LIN {X 0,Y 450.546,Z 601.299,A -85,B 0,C 180,E1 -16151.951,E2 -16151.951} C_VEL
LIN {X 0,Y 450.573,Z 601.291,A -85,B 0,C 180,E1 -16154.391,E2 -16154.391} C_VEL
LIN {X 0,Y 450.568,Z 601.288,A -85,B 0,C 180,E1 -16156.941,E2 -16156.941} C_VEL
LIN {X 0,Y 450.573,Z 601.291,A -85,B 0,C 180,E1 -16160.405,E2 -16160.405} C_VEL
LIN {X 0,Y 450.592,Z 601.291,A -85,B 0,C 180,E1 -16163.793,E2 -16163.793} C_VEL
LIN {X 0,Y 450.566,Z 601.289,A -85,B 0,C 180,E1 -16167.085,E2 -16167.085} C_VEL
LIN {X 0,Y 450.558,Z 601.295,A -85,B 0,C 180,E1 -16170.167,E2 -16170.167} C_VEL
LIN {X 0,Y 450.589,Z 601.286,A -85,B 0,C 180,E1 -16173.205,E2 -16173.205} C_VEL
LIN {X 0,Y 450.58,Z 601.289,A -85,B 0,C 180,E1 -16176.517,E2 -16176.517} C_VEL
LIN {X 0,Y 450.593,Z 601.293,A -85,B 0,C 180,E1 -16180.002,E2 -16180.002} C_VEL
LIN {X 0,Y 450.589,Z 601.286,A -85,B 0,C 180,E1 -16182.821,E2 -16182.821} C_VEL
LIN {X 0,Y 450.626,Z 601.284,A -85,B 0,C 180,E1 -16185.6,E2 -16185.6} C_VEL
LIN {X 0,Y 450.749,Z 601.269,A -85,B 0,C 180,E1 -16188.346,E2 -16188.346} C_VEL
LIN {X 0,Y 450.78,Z 601.27,A -85,B 0,C 180,E1 -16191.961,E2 -16191.961} C_VEL
LIN {X 0,Y 450.913,Z 601.251,A -85,B 0,C 180,E1 -16193.81,E2 -16193.81} C_VEL
LIN {X 0,Y 450.837,Z 601.258,A -85,B 0,C 180,E1 -16196.437,E2 -16196.437} C_VEL
LIN {X 0,Y 450.905,Z 601.254,A -85,B 0,C 180,E1 -16200,E2 -16200} C_VEL
LIN {X 0,Y 450.866,Z 601.254,A -85,B 0,C 180,E1 -16204.455,E2 -16204.455} C_VEL
LIN {X 0,Y 450.774,Z 601.263,A -85,B 0,C 180,E1 -16207.141,E2 -16207.141} C_VEL
LIN {X 0,Y 450.679,Z 601.281,A -85,B 0,C 180,E1 -16209.844,E2 -16209.844} C_VEL
LIN {X 0,Y 450.674,Z 601.277,A -85,B 0,C 180,E1 -16212.568,E2 -16212.568} C_VEL
LIN {X 0,Y 450.622,Z 601.284,A -85,B 0,C 180,E1 -16215.48,E2 -16215.48} C_VEL
LIN {X 0,Y 450.567,Z 601.289,A -85,B 0,C 180,E1 -16219.054,E2 -16219.054} C_VEL
LIN {X 0,Y 450.548,Z 601.298,A -85,B 0,C 180,E1 -16221.908,E2 -16221.908} C_VEL
LIN {X 0,Y 450.531,Z 601.293,A -85,B 0,C 180,E1 -16224.82,E2 -16224.82} C_VEL
LIN {X 0,Y 450.577,Z 601.293,A -85,B 0,C 180,E1 -16227.799,E2 -16227.799} C_VEL
LIN {X 0,Y 450.517,Z 601.295,A -85,B 0,C 180,E1 -16230.869,E2 -16230.869} C_VEL
LIN {X 0,Y 450.532,Z 601.3,A -85,B 0,C 180,E1 -16234.035,E2 -16234.035} C_VEL
LIN {X 0,Y 450.534,Z 601.298,A -85,B 0,C 180,E1 -16236.213,E2 -16236.213} C_VEL
LIN {X 0,Y 450.5,Z 601.3,A -85,B 0,C 180,E1 -16239.604,E2 -16239.604} C_VEL
LIN {X 0,Y 450.53,Z 601.301,A -85,B 0,C 180,E1 -16241.953,E2 -16241.953} C_VEL
LIN {X 0,Y 450.556,Z 601.293,A -85,B 0,C 180,E1 -16244.393,E2 -16244.393} C_VEL
LIN {X 0,Y 450.538,Z 601.292,A -85,B 0,C 180,E1 -16246.945,E2 -16246.945} C_VEL
LIN {X 0,Y 450.509,Z 601.299,A -85,B 0,C 180,E1 -16249.627,E2 -16249.627} C_VEL
LIN {X 0,Y 450.48,Z 601.3,A -85,B 0,C 180,E1 -16252.67,E2 -16252.67} C_VEL
LIN {X 0,Y 450.521,Z 601.302,A -85,B 0,C 180,E1 -16255.965,E2 -16255.965} C_VEL
LIN {X 0,Y 450.517,Z 601.295,A -85,B 0,C 180,E1 -16259.132,E2 -16259.132} C_VEL
LIN {X 0,Y 450.547,Z 601.291,A -85,B 0,C 180,E1 -16261.188,E2 -16261.188} C_VEL
LIN {X 0,Y 450.616,Z 601.459,A -85,B 0,C 180,E1 -16264.463,E2 -16264.463} C_VEL
LIN {X 0,Y 453.094,Z 615.734,A -85,B 0,C 180,E1 -16267.528,E2 -16267.528} C_VEL
LIN {X 0,Y 452.123,Z 628.307,A -85,B 0,C 180,E1 -16270.073,E2 -16270.073} C_VEL
LIN {X 0,Y 450.856,Z 645.268,A -85,B 0,C 180,E1 -16273.471,E2 -16273.471} C_VEL
LIN {X 0,Y 453.98,Z 674.168,A -85,B 0,C 180,E1 -16274.153,E2 -16274.153} C_VEL
LIN {X 0,Y 454.049,Z 687.401,A -85,B 0,C 180,E1 -16274.424,E2 -16274.424} C_VEL
LIN {X 0,Y 452.771,Z 752.366,A -85,B 0,C 180,E1 -16275.726,E2 -16275.726} C_VEL
LIN {X 0,Y 452.55,Z 762.586,A -85,B 0,C 180,E1 -16276.034,E2 -16276.034} C_VEL
LIN {X 0,Y 452.15,Z 772.789,A -85,B 0,C 180,E1 -16276.449,E2 -16276.449} C_VEL
LIN {X 0,Y 451.855,Z 781.497,A -85,B 0,C 180,E1 -16276.897,E2 -16276.897} C_VEL
LIN {X 0,Y 451.313,Z 791.921,A -85,B 0,C 180,E1 -16277.565,E2 -16277.565} C_VEL
LIN {X 0,Y 450.749,Z 801.808,A -85,B 0,C 180,E1 -16278.345,E2 -16278.345} C_VEL
LIN {X 0,Y 450.383,Z 810.122,A -85,B 0,C 180,E1 -16279.131,E2 -16279.131} C_VEL
LIN {X 0,Y 449.846,Z 819.008,A -85,B 0,C 180,E1 -16280.138,E2 -16280.138} C_VEL
LIN {X 0,Y 449.477,Z 825.737,A -85,B 0,C 180,E1 -16281.035,E2 -16281.035} C_VEL
LIN {X 0,Y 449.096,Z 832.781,A -85,B 0,C 180,E1 -16282.156,E2 -16282.156} C_VEL
LIN {X 0,Y 448.876,Z 838.658,A -85,B 0,C 180,E1 -16283.279,E2 -16283.279} C_VEL
LIN {X 0,Y 448.702,Z 844.329,A -85,B 0,C 180,E1 -16284.626,E2 -16284.626} C_VEL
LIN {X 0,Y 448.577,Z 848.751,A -85,B 0,C 180,E1 -16285.971,E2 -16285.971} C_VEL
LIN {X 0,Y 448.542,Z 852.046,A -85,B 0,C 180,E1 -16287.315,E2 -16287.315} C_VEL
LIN {X 0,Y 448.542,Z 853.712,A -85,B 0,C 180,E1 -16288.21,E2 -16288.21} C_VEL
LIN {X 0,Y 448.535,Z 855.564,A -85,B 0,C 180,E1 -16290,E2 -16290} C_VEL
LIN {X 0,Y 448.515,Z 855.863,A -85,B 0,C 180,E1 -16290.895,E2 -16290.895} C_VEL
LIN {X 0,Y 448.491,Z 855.194,A -85,B 0,C 180,E1 -16292.686,E2 -16292.686} C_VEL
LIN {X 0,Y 448.542,Z 854.146,A -85,B 0,C 180,E1 -16293.581,E2 -16293.581} C_VEL
LIN {X 0,Y 448.749,Z 850.921,A -85,B 0,C 180,E1 -16295.374,E2 -16295.374} C_VEL
LIN {X 0,Y 449.026,Z 847.231,A -85,B 0,C 180,E1 -16296.719,E2 -16296.719} C_VEL
LIN {X 0,Y 449.487,Z 842.395,A -85,B 0,C 180,E1 -16298.062,E2 -16298.062} C_VEL
LIN {X 0,Y 450.082,Z 836.291,A -85,B 0,C 180,E1 -16299.405,E2 -16299.405} C_VEL
LIN {X 0,Y 450.945,Z 828.69,A -85,B 0,C 180,E1 -16300.743,E2 -16300.743} C_VEL
LIN {X 0,Y 451.886,Z 821.013,A -85,B 0,C 180,E1 -16301.852,E2 -16301.852} C_VEL
LIN {X 0,Y 452.624,Z 813.883,A -85,B 0,C 180,E1 -16302.731,E2 -16302.731} C_VEL
LIN {X 0,Y 453.681,Z 804.065,A -85,B 0,C 180,E1 -16303.732,E2 -16303.732} C_VEL
LIN {X 0,Y 454.54,Z 795.005,A -85,B 0,C 180,E1 -16304.502,E2 -16304.502} C_VEL
LIN {X 0,Y 455.414,Z 785.704,A -85,B 0,C 180,E1 -16305.157,E2 -16305.157} C_VEL
LIN {X 0,Y 456.23,Z 775.218,A -85,B 0,C 180,E1 -16305.757,E2 -16305.757} C_VEL
LIN {X 0,Y 457.128,Z 763.471,A -85,B 0,C 180,E1 -16306.267,E2 -16306.267} C_VEL
LIN {X 0,Y 457.765,Z 752.645,A -85,B 0,C 180,E1 -16306.616,E2 -16306.616} C_VEL
LIN {X 0,Y 458.823,Z 722.033,A -85,B 0,C 180,E1 -16307.29,E2 -16307.29} C_VEL
LIN {X 0,Y 460.202,Z 677.981,A -85,B 0,C 180,E1 -16308.254,E2 -16308.254} C_VEL
LIN {X 0,Y 457.656,Z 661.739,A -85,B 0,C 180,E1 -16308.813,E2 -16308.813} C_VEL
LIN {X 0,Y 454.289,Z 646.219,A -85,B 0,C 180,E1 -16309.435,E2 -16309.435} C_VEL
LIN {X 0,Y 453.659,Z 643.473,A -85,B 0,C 180,E1 -16309.562,E2 -16309.562} C_VEL
LIN {X 0,Y 455.818,Z 627.583,A -85,B 0,C 180,E1 -16313.07,E2 -16313.07} C_VEL
LIN {X 0,Y 454.965,Z 621.055,A -85,B 0,C 180,E1 -16314.723,E2 -16314.723} C_VEL
LIN {X 0,Y 453.262,Z 612.283,A -85,B 0,C 180,E1 -16317.122,E2 -16317.122} C_VEL
LIN {X 0,Y 451.108,Z 603.423,A -85,B 0,C 180,E1 -16319.793,E2 -16319.793} C_VEL
LIN {X 0,Y 450.552,Z 601.297,A -85,B 0,C 180,E1 -16320.478,E2 -16320.478} C_VEL
LIN {X 0,Y 450.545,Z 601.297,A -85,B 0,C 180,E1 -16324.034,E2 -16324.034} C_VEL
LIN {X 0,Y 450.52,Z 601.296,A -85,B 0,C 180,E1 -16327.326,E2 -16327.326} C_VEL
LIN {X 0,Y 450.53,Z 601.291,A -85,B 0,C 180,E1 -16330.376,E2 -16330.376} C_VEL
LIN {X 0,Y 450.55,Z 601.291,A -85,B 0,C 180,E1 -16333.161,E2 -16333.161} C_VEL
LIN {X 0,Y 450.576,Z 601.291,A -85,B 0,C 180,E1 -16335.651,E2 -16335.651} C_VEL
LIN {X 0,Y 450.551,Z 601.296,A -85,B 0,C 180,E1 -16338.265,E2 -16338.265} C_VEL
LIN {X 0,Y 450.564,Z 601.292,A -85,B 0,C 180,E1 -16341.014,E2 -16341.014} C_VEL
LIN {X 0,Y 450.555,Z 601.294,A -85,B 0,C 180,E1 -16343.941,E2 -16343.941} C_VEL
LIN {X 0,Y 450.579,Z 601.295,A -85,B 0,C 180,E1 -16347.083,E2 -16347.083} C_VEL
LIN {X 0,Y 450.562,Z 601.292,A -85,B 0,C 180,E1 -16350.167,E2 -16350.167} C_VEL
LIN {X 0,Y 450.602,Z 601.289,A -85,B 0,C 180,E1 -16353.205,E2 -16353.205} C_VEL
LIN {X 0,Y 450.584,Z 601.295,A -85,B 0,C 180,E1 -16356.517,E2 -16356.517} C_VEL
LIN {X 0,Y 450.597,Z 601.297,A -85,B 0,C 180,E1 -16360.002,E2 -16360.002} C_VEL
LIN {X 0,Y 450.61,Z 601.344,A -85,B 0,C 180,E1 -16362.589,E2 -16362.589} C_VEL
LIN {X 0,Y 452.468,Z 609.128,A -85,B 0,C 180,E1 -16365.201,E2 -16365.201} C_VEL
LIN {X 0,Y 454.016,Z 616.689,A -85,B 0,C 180,E1 -16367.526,E2 -16367.526} C_VEL
LIN {X 0,Y 454.947,Z 623.05,A -85,B 0,C 180,E1 -16369.353,E2 -16369.353} C_VEL
LIN {X 0,Y 454.575,Z 627.715,A -85,B 0,C 180,E1 -16370.56,E2 -16370.56} C_VEL
LIN {X 0,Y 459.098,Z 645.694,A -85,B 0,C 180,E1 -16371.343,E2 -16371.343} C_VEL
LIN {X 0,Y 460.909,Z 655.517,A -85,B 0,C 180,E1 -16371.699,E2 -16371.699} C_VEL
LIN {X 0,Y 458.567,Z 715.512,A -85,B 0,C 180,E1 -16372.981,E2 -16372.981} C_VEL
LIN {X 0,Y 457.808,Z 737.352,A -85,B 0,C 180,E1 -16373.493,E2 -16373.493} C_VEL
LIN {X 0,Y 457.027,Z 751.138,A -85,B 0,C 180,E1 -16374.007,E2 -16374.007} C_VEL
LIN {X 0,Y 456.261,Z 762.657,A -85,B 0,C 180,E1 -16374.604,E2 -16374.604} C_VEL
LIN {X 0,Y 455.54,Z 772.672,A -85,B 0,C 180,E1 -16375.259,E2 -16375.259} C_VEL
LIN {X 0,Y 454.727,Z 782.259,A -85,B 0,C 180,E1 -16376.025,E2 -16376.025} C_VEL
LIN {X 0,Y 453.809,Z 791.383,A -85,B 0,C 180,E1 -16376.903,E2 -16376.903} C_VEL
LIN {X 0,Y 452.94,Z 799.112,A -85,B 0,C 180,E1 -16377.784,E2 -16377.784} C_VEL
LIN {X 0,Y 451.916,Z 807.198,A -85,B 0,C 180,E1 -16378.89,E2 -16378.89} C_VEL
LIN {X 0,Y 451.029,Z 813.945,A -85,B 0,C 180,E1 -16380,E2 -16380} C_VEL
LIN {X 0,Y 450.508,Z 818.593,A -85,B 0,C 180,E1 -16380.891,E2 -16380.891} C_VEL
LIN {X 0,Y 449.775,Z 824.257,A -85,B 0,C 180,E1 -16382.231,E2 -16382.231} C_VEL
LIN {X 0,Y 449.416,Z 828.692,A -85,B 0,C 180,E1 -16383.574,E2 -16383.574} C_VEL
LIN {X 0,Y 449.156,Z 831.048,A -85,B 0,C 180,E1 -16384.472,E2 -16384.472} C_VEL
LIN {X 0,Y 448.716,Z 834.413,A -85,B 0,C 180,E1 -16386.273,E2 -16386.273} C_VEL
LIN {X 0,Y 448.549,Z 835.387,A -85,B 0,C 180,E1 -16387.176,E2 -16387.176} C_VEL
LIN {X 0,Y 448.418,Z 836.149,A -85,B 0,C 180,E1 -16388.986,E2 -16388.986} C_VEL
LIN {X 0,Y 448.466,Z 835.598,A -85,B 0,C 180,E1 -16390.269,E2 -16390.269} C_VEL
LIN {X 0,Y 448.381,Z 833.919,A -85,B 0,C 180,E1 -16391.717,E2 -16391.717} C_VEL
LIN {X 0,Y 448.492,Z 831.264,A -85,B 0,C 180,E1 -16393.088,E2 -16393.088} C_VEL
LIN {X 0,Y 448.702,Z 827.132,A -85,B 0,C 180,E1 -16394.567,E2 -16394.567} C_VEL
LIN {X 0,Y 448.922,Z 821.42,A -85,B 0,C 180,E1 -16396.078,E2 -16396.078} C_VEL
LIN {X 0,Y 449.14,Z 815.962,A -85,B 0,C 180,E1 -16397.236,E2 -16397.236} C_VEL
LIN {X 0,Y 449.473,Z 809.329,A -85,B 0,C 180,E1 -16398.395,E2 -16398.395} C_VEL
LIN {X 0,Y 449.829,Z 803.085,A -85,B 0,C 180,E1 -16399.322,E2 -16399.322} C_VEL
LIN {X 0,Y 450.304,Z 793.566,A -85,B 0,C 180,E1 -16400.486,E2 -16400.486} C_VEL
LIN {X 0,Y 450.736,Z 784.964,A -85,B 0,C 180,E1 -16401.362,E2 -16401.362} C_VEL
LIN {X 0,Y 451.211,Z 776.182,A -85,B 0,C 180,E1 -16402.113,E2 -16402.113} C_VEL
LIN {X 0,Y 451.7,Z 766.35,A -85,B 0,C 180,E1 -16402.809,E2 -16402.809} C_VEL
LIN {X 0,Y 452.132,Z 756.214,A -85,B 0,C 180,E1 -16403.389,E2 -16403.389} C_VEL
LIN {X 0,Y 452.394,Z 745.054,A -85,B 0,C 180,E1 -16403.886,E2 -16403.886} C_VEL
LIN {X 0,Y 452.747,Z 734.354,A -85,B 0,C 180,E1 -16404.235,E2 -16404.235} C_VEL
LIN {X 0,Y 453.276,Z 712.839,A -85,B 0,C 180,E1 -16404.69,E2 -16404.69} C_VEL
LIN {X 0,Y 454.432,Z 650.819,A -85,B 0,C 180,E1 -16405.918,E2 -16405.918} C_VEL
LIN {X 0,Y 451.139,Z 625.367,A -85,B 0,C 180,E1 -16406.542,E2 -16406.542} C_VEL
LIN {X 0,Y 452.027,Z 612.321,A -85,B 0,C 180,E1 -16409.471,E2 -16409.471} C_VEL
LIN {X 0,Y 451.77,Z 607.809,A -85,B 0,C 180,E1 -16410.515,E2 -16410.515} C_VEL
LIN {X 0,Y 450.631,Z 601.287,A -85,B 0,C 180,E1 -16412.099,E2 -16412.099} C_VEL
LIN {X 0,Y 450.56,Z 601.289,A -85,B 0,C 180,E1 -16415.113,E2 -16415.113} C_VEL
LIN {X 0,Y 450.547,Z 601.293,A -85,B 0,C 180,E1 -16418.451,E2 -16418.451} C_VEL
LIN {X 0,Y 450.55,Z 601.291,A -85,B 0,C 180,E1 -16420.764,E2 -16420.764} C_VEL
LIN {X 0,Y 450.57,Z 601.288,A -85,B 0,C 180,E1 -16423.157,E2 -16423.157} C_VEL
LIN {X 0,Y 450.574,Z 601.291,A -85,B 0,C 180,E1 -16425.65,E2 -16425.65} C_VEL
LIN {X 0,Y 450.548,Z 601.295,A -85,B 0,C 180,E1 -16428.264,E2 -16428.264} C_VEL
LIN {X 0,Y 450.561,Z 601.289,A -85,B 0,C 180,E1 -16431.013,E2 -16431.013} C_VEL
LIN {X 0,Y 450.578,Z 601.295,A -85,B 0,C 180,E1 -16433.935,E2 -16433.935} C_VEL
LIN {X 0,Y 450.566,Z 601.289,A -85,B 0,C 180,E1 -16437.084,E2 -16437.084} C_VEL
LIN {X 0,Y 450.577,Z 601.289,A -85,B 0,C 180,E1 -16440.521,E2 -16440.521} C_VEL
LIN {X 0,Y 450.588,Z 601.286,A -85,B 0,C 180,E1 -16443.204,E2 -16443.204} C_VEL
LIN {X 0,Y 450.578,Z 601.289,A -85,B 0,C 180,E1 -16446.516,E2 -16446.516} C_VEL
LIN {X 0,Y 450.591,Z 601.294,A -85,B 0,C 180,E1 -16450.002,E2 -16450.002} C_VEL
LIN {X 0,Y 450.604,Z 601.284,A -85,B 0,C 180,E1 -16452.821,E2 -16452.821} C_VEL
LIN {X 0,Y 450.66,Z 601.28,A -85,B 0,C 180,E1 -16455.6,E2 -16455.6} C_VEL
LIN {X 0,Y 450.745,Z 601.27,A -85,B 0,C 180,E1 -16458.345,E2 -16458.345} C_VEL
LIN {X 0,Y 450.776,Z 601.27,A -85,B 0,C 180,E1 -16461.961,E2 -16461.961} C_VEL
LIN {X 0,Y 450.824,Z 601.257,A -85,B 0,C 180,E1 -16464.651,E2 -16464.651} C_VEL
LIN {X 0,Y 450.722,Z 601.27,A -85,B 0,C 180,E1 -16467.328,E2 -16467.328} C_VEL
LIN {X 0,Y 450.902,Z 601.255,A -85,B 0,C 180,E1 -16470,E2 -16470} C_VEL
LIN {X 0,Y 450.873,Z 601.253,A -85,B 0,C 180,E1 -16474.455,E2 -16474.455} C_VEL
LIN {X 0,Y 450.769,Z 601.263,A -85,B 0,C 180,E1 -16477.141,E2 -16477.141} C_VEL
LIN {X 0,Y 450.675,Z 601.281,A -85,B 0,C 180,E1 -16479.844,E2 -16479.844} C_VEL
LIN {X 0,Y 450.69,Z 601.275,A -85,B 0,C 180,E1 -16482.567,E2 -16482.567} C_VEL
LIN {X 0,Y 450.7,Z 601.274,A -85,B 0,C 180,E1 -16485.518,E2 -16485.518} C_VEL
LIN {X 0,Y 450.584,Z 601.286,A -85,B 0,C 180,E1 -16489.053,E2 -16489.053} C_VEL
LIN {X 0,Y 450.574,Z 601.294,A -85,B 0,C 180,E1 -16491.906,E2 -16491.906} C_VEL
LIN {X 0,Y 450.53,Z 601.293,A -85,B 0,C 180,E1 -16494.82,E2 -16494.82} C_VEL
LIN {X 0,Y 450.576,Z 601.293,A -85,B 0,C 180,E1 -16497.798,E2 -16497.798} C_VEL
LIN {X 0,Y 450.592,Z 601.285,A -85,B 0,C 180,E1 -16500.863,E2 -16500.863} C_VEL
LIN {X 0,Y 450.583,Z 601.294,A -85,B 0,C 180,E1 -16504.03,E2 -16504.03} C_VEL
LIN {X 0,Y 450.604,Z 601.29,A -85,B 0,C 180,E1 -16506.106,E2 -16506.106} C_VEL
LIN {X 0,Y 449.93,Z 601.37,A -85,B 0,C 180,E1 -16506.851,E2 -16506.851} C_VEL
LIN {X 0,Y 447.042,Z 601.735,A -85,B 0,C 180,E1 -16508.061,E2 -16508.061} C_VEL
LIN {X 0,Y 444.609,Z 602.033,A -85,B 0,C 180,E1 -16509.037,E2 -16509.037} C_VEL
LIN {X 0,Y 443.58,Z 602.164,A -85,B 0,C 180,E1 -16509.792,E2 -16509.792} C_VEL
LIN {X 0,Y 443.505,Z 602.169,A -85,B 0,C 180,E1 -16510.047,E2 -16510.047} C_VEL
LIN {X 0,Y 443.516,Z 602.168,A -85,B 0,C 180,E1 -16513.409,E2 -16513.409} C_VEL
LIN {X 0,Y 443.516,Z 602.168,A -85,B 0,C 180,E1 -16516.592,E2 -16516.592} C_VEL
LIN {X 0,Y 443.521,Z 602.17,A -85,B 0,C 180,E1 -16519.647,E2 -16519.647} C_VEL
LIN {X 0,Y 443.527,Z 602.171,A -85,B 0,C 180,E1 -16522.151,E2 -16522.151} C_VEL
LIN {X 0,Y 443.526,Z 602.167,A -85,B 0,C 180,E1 -16525.352,E2 -16525.352} C_VEL
LIN {X 0,Y 443.534,Z 602.166,A -85,B 0,C 180,E1 -16528.591,E2 -16528.591} C_VEL
LIN {X 0,Y 443.521,Z 602.171,A -85,B 0,C 180,E1 -16531.72,E2 -16531.72} C_VEL
LIN {X 0,Y 443.491,Z 602.17,A -85,B 0,C 180,E1 -16534.759,E2 -16534.759} C_VEL
LIN {X 0,Y 443.509,Z 602.172,A -85,B 0,C 180,E1 -16537.726,E2 -16537.726} C_VEL
LIN {X 0,Y 443.557,Z 602.163,A -85,B 0,C 180,E1 -16540.633,E2 -16540.633} C_VEL
LIN {X 0,Y 443.555,Z 602.164,A -85,B 0,C 180,E1 -16543.486,E2 -16543.486} C_VEL
LIN {X 0,Y 443.593,Z 602.161,A -85,B 0,C 180,E1 -16546.299,E2 -16546.299} C_VEL
LIN {X 0,Y 443.665,Z 602.148,A -85,B 0,C 180,E1 -16549.08,E2 -16549.08} C_VEL
LIN {X 0,Y 443.777,Z 602.135,A -85,B 0,C 180,E1 -16552.746,E2 -16552.746} C_VEL
LIN {X 0,Y 443.843,Z 602.128,A -85,B 0,C 180,E1 -16555.475,E2 -16555.475} C_VEL
LIN {X 0,Y 443.858,Z 602.132,A -85,B 0,C 180,E1 -16560,E2 -16560} C_VEL
LIN {X 0,Y 443.837,Z 602.129,A -85,B 0,C 180,E1 -16564.526,E2 -16564.526} C_VEL
LIN {X 0,Y 443.749,Z 602.138,A -85,B 0,C 180,E1 -16567.255,E2 -16567.255} C_VEL
LIN {X 0,Y 443.659,Z 602.149,A -85,B 0,C 180,E1 -16570.921,E2 -16570.921} C_VEL
LIN {X 0,Y 443.588,Z 602.162,A -85,B 0,C 180,E1 -16573.701,E2 -16573.701} C_VEL
LIN {X 0,Y 443.519,Z 602.168,A -85,B 0,C 180,E1 -16576.516,E2 -16576.516} C_VEL
LIN {X 0,Y 443.509,Z 602.169,A -85,B 0,C 180,E1 -16579.37,E2 -16579.37} C_VEL
LIN {X 0,Y 443.491,Z 602.174,A -85,B 0,C 180,E1 -16582.275,E2 -16582.275} C_VEL
LIN {X 0,Y 443.487,Z 602.171,A -85,B 0,C 180,E1 -16585.242,E2 -16585.242} C_VEL
LIN {X 0,Y 443.519,Z 602.171,A -85,B 0,C 180,E1 -16588.28,E2 -16588.28} C_VEL
LIN {X 0,Y 443.481,Z 602.173,A -85,B 0,C 180,E1 -16591.473,E2 -16591.473} C_VEL
LIN {X 0,Y 443.49,Z 602.17,A -85,B 0,C 180,E1 -16594.787,E2 -16594.787} C_VEL
LIN {X 0,Y 443.482,Z 602.179,A -85,B 0,C 180,E1 -16598.023,E2 -16598.023} C_VEL
LIN {X 0,Y 443.483,Z 602.174,A -85,B 0,C 180,E1 -16601.556,E2 -16601.556} C_VEL
LIN {X 0,Y 443.492,Z 602.171,A -85,B 0,C 180,E1 -16604.706,E2 -16604.706} C_VEL
LIN {X 0,Y 443.489,Z 602.177,A -85,B 0,C 180,E1 -16607.929,E2 -16607.929} C_VEL
LIN {X 0,Y 443.48,Z 602.172,A -85,B 0,C 180,E1 -16610.819,E2 -16610.819} C_VEL
LIN {X 0,Y 443.464,Z 602.178,A -85,B 0,C 180,E1 -16614.239,E2 -16614.239} C_VEL
LIN {X 0,Y 443.472,Z 602.175,A -85,B 0,C 180,E1 -16617.519,E2 -16617.519} C_VEL
LIN {X 0,Y 443.523,Z 602.167,A -85,B 0,C 180,E1 -16620.688,E2 -16620.688} C_VEL
LIN {X 0,Y 443.572,Z 602.266,A -85,B 0,C 180,E1 -16624.342,E2 -16624.342} C_VEL
LIN {X 0,Y 446.022,Z 616.142,A -85,B 0,C 180,E1 -16627.372,E2 -16627.372} C_VEL
LIN {X 0,Y 445.295,Z 626.543,A -85,B 0,C 180,E1 -16629.513,E2 -16629.513} C_VEL
LIN {X 0,Y 443.844,Z 645.08,A -85,B 0,C 180,E1 -16633.291,E2 -16633.291} C_VEL
LIN {X 0,Y 446.963,Z 674.631,A -85,B 0,C 180,E1 -16634.004,E2 -16634.004} C_VEL
LIN {X 0,Y 447.101,Z 684.625,A -85,B 0,C 180,E1 -16634.217,E2 -16634.217} C_VEL
LIN {X 0,Y 445.784,Z 751.209,A -85,B 0,C 180,E1 -16635.585,E2 -16635.585} C_VEL
LIN {X 0,Y 445.524,Z 761.668,A -85,B 0,C 180,E1 -16635.896,E2 -16635.896} C_VEL
LIN {X 0,Y 445.165,Z 771.447,A -85,B 0,C 180,E1 -16636.291,E2 -16636.291} C_VEL
LIN {X 0,Y 444.799,Z 781.293,A -85,B 0,C 180,E1 -16636.801,E2 -16636.801} C_VEL
LIN {X 0,Y 444.251,Z 792.006,A -85,B 0,C 180,E1 -16637.502,E2 -16637.502} C_VEL
LIN {X 0,Y 443.716,Z 801.029,A -85,B 0,C 180,E1 -16638.222,E2 -16638.222} C_VEL
LIN {X 0,Y 443.323,Z 809.905,A -85,B 0,C 180,E1 -16639.071,E2 -16639.071} C_VEL
LIN {X 0,Y 442.805,Z 817.917,A -85,B 0,C 180,E1 -16639.98,E2 -16639.98} C_VEL
LIN {X 0,Y 442.332,Z 826.248,A -85,B 0,C 180,E1 -16641.119,E2 -16641.119} C_VEL
LIN {X 0,Y 441.989,Z 833.181,A -85,B 0,C 180,E1 -16642.259,E2 -16642.259} C_VEL
LIN {X 0,Y 441.821,Z 837.963,A -85,B 0,C 180,E1 -16643.171,E2 -16643.171} C_VEL
LIN {X 0,Y 441.62,Z 843.753,A -85,B 0,C 180,E1 -16644.539,E2 -16644.539} C_VEL
LIN {X 0,Y 441.502,Z 848.278,A -85,B 0,C 180,E1 -16645.906,E2 -16645.906} C_VEL
LIN {X 0,Y 441.459,Z 851.667,A -85,B 0,C 180,E1 -16647.272,E2 -16647.272} C_VEL
LIN {X 0,Y 441.454,Z 853.695,A -85,B 0,C 180,E1 -16648.387,E2 -16648.387} C_VEL
LIN {X 0,Y 441.456,Z 855.355,A -85,B 0,C 180,E1 -16650,E2 -16650} C_VEL
LIN {X 0,Y 441.398,Z 855.734,A -85,B 0,C 180,E1 -16651.33,E2 -16651.33} C_VEL
LIN {X 0,Y 441.396,Z 855.12,A -85,B 0,C 180,E1 -16652.729,E2 -16652.729} C_VEL
LIN {X 0,Y 441.523,Z 852.715,A -85,B 0,C 180,E1 -16654.55,E2 -16654.55} C_VEL
LIN {X 0,Y 441.76,Z 849.815,A -85,B 0,C 180,E1 -16655.916,E2 -16655.916} C_VEL
LIN {X 0,Y 442.092,Z 845.859,A -85,B 0,C 180,E1 -16657.282,E2 -16657.282} C_VEL
LIN {X 0,Y 442.47,Z 842.664,A -85,B 0,C 180,E1 -16658.191,E2 -16658.191} C_VEL
LIN {X 0,Y 443.194,Z 835.505,A -85,B 0,C 180,E1 -16659.782,E2 -16659.782} C_VEL
LIN {X 0,Y 443.995,Z 829.216,A -85,B 0,C 180,E1 -16660.913,E2 -16660.913} C_VEL
LIN {X 0,Y 444.979,Z 821.66,A -85,B 0,C 180,E1 -16662.039,E2 -16662.039} C_VEL
LIN {X 0,Y 445.889,Z 813.574,A -85,B 0,C 180,E1 -16663.05,E2 -16663.05} C_VEL
LIN {X 0,Y 446.972,Z 803.798,A -85,B 0,C 180,E1 -16664.058,E2 -16664.058} C_VEL
LIN {X 0,Y 447.888,Z 794.746,A -85,B 0,C 180,E1 -16664.838,E2 -16664.838} C_VEL
LIN {X 0,Y 448.802,Z 785.52,A -85,B 0,C 180,E1 -16665.502,E2 -16665.502} C_VEL
LIN {X 0,Y 449.675,Z 775.152,A -85,B 0,C 180,E1 -16666.109,E2 -16666.109} C_VEL
LIN {X 0,Y 450.64,Z 763.575,A -85,B 0,C 180,E1 -16666.624,E2 -16666.624} C_VEL
LIN {X 0,Y 451.285,Z 752.987,A -85,B 0,C 180,E1 -16666.977,E2 -16666.977} C_VEL
LIN {X 0,Y 452.121,Z 730.269,A -85,B 0,C 180,E1 -16667.497,E2 -16667.497} C_VEL
LIN {X 0,Y 453.848,Z 679.041,A -85,B 0,C 180,E1 -16668.635,E2 -16668.635} C_VEL
LIN {X 0,Y 451.412,Z 663.155,A -85,B 0,C 180,E1 -16669.204,E2 -16669.204} C_VEL
LIN {X 0,Y 447.884,Z 647.11,A -85,B 0,C 180,E1 -16669.878,E2 -16669.878} C_VEL
LIN {X 0,Y 447.032,Z 643.209,A -85,B 0,C 180,E1 -16670.066,E2 -16670.066} C_VEL
LIN {X 0,Y 449.014,Z 629.365,A -85,B 0,C 180,E1 -16673.197,E2 -16673.197} C_VEL
LIN {X 0,Y 448.121,Z 622.532,A -85,B 0,C 180,E1 -16674.963,E2 -16674.963} C_VEL
LIN {X 0,Y 446.283,Z 613.275,A -85,B 0,C 180,E1 -16677.581,E2 -16677.581} C_VEL
LIN {X 0,Y 444.14,Z 604.6,A -85,B 0,C 180,E1 -16680.309,E2 -16680.309} C_VEL
LIN {X 0,Y 443.502,Z 602.177,A -85,B 0,C 180,E1 -16681.147,E2 -16681.147} C_VEL
LIN {X 0,Y 443.529,Z 602.169,A -85,B 0,C 180,E1 -16684.794,E2 -16684.794} C_VEL
LIN {X 0,Y 443.493,Z 602.165,A -85,B 0,C 180,E1 -16688.022,E2 -16688.022} C_VEL
LIN {X 0,Y 443.49,Z 602.167,A -85,B 0,C 180,E1 -16691.556,E2 -16691.556} C_VEL
LIN {X 0,Y 443.513,Z 602.172,A -85,B 0,C 180,E1 -16694.709,E2 -16694.709} C_VEL
LIN {X 0,Y 443.508,Z 602.174,A -85,B 0,C 180,E1 -16697.927,E2 -16697.927} C_VEL
LIN {X 0,Y 443.531,Z 602.168,A -85,B 0,C 180,E1 -16700.824,E2 -16700.824} C_VEL
LIN {X 0,Y 443.504,Z 602.172,A -85,B 0,C 180,E1 -16704.242,E2 -16704.242} C_VEL
LIN {X 0,Y 443.532,Z 602.169,A -85,B 0,C 180,E1 -16707.524,E2 -16707.524} C_VEL
LIN {X 0,Y 443.535,Z 602.172,A -85,B 0,C 180,E1 -16710.688,E2 -16710.688} C_VEL
LIN {X 0,Y 443.556,Z 602.168,A -85,B 0,C 180,E1 -16714.174,E2 -16714.174} C_VEL
LIN {X 0,Y 443.538,Z 602.173,A -85,B 0,C 180,E1 -16716.746,E2 -16716.746} C_VEL
LIN {X 0,Y 443.548,Z 602.173,A -85,B 0,C 180,E1 -16719.67,E2 -16719.67} C_VEL
LIN {X 0,Y 443.604,Z 602.207,A -85,B 0,C 180,E1 -16721.948,E2 -16721.948} C_VEL
LIN {X 0,Y 445.657,Z 610.9,A -85,B 0,C 180,E1 -16724.969,E2 -16724.969} C_VEL
LIN {X 0,Y 447.175,Z 618.363,A -85,B 0,C 180,E1 -16727.332,E2 -16727.332} C_VEL
LIN {X 0,Y 448.139,Z 624.657,A -85,B 0,C 180,E1 -16729.189,E2 -16729.189} C_VEL
LIN {X 0,Y 447.971,Z 628.17,A -85,B 0,C 180,E1 -16730.086,E2 -16730.086} C_VEL
LIN {X 0,Y 452.991,Z 647.727,A -85,B 0,C 180,E1 -16730.971,E2 -16730.971} C_VEL
LIN {X 0,Y 454.591,Z 656.836,A -85,B 0,C 180,E1 -16731.318,E2 -16731.318} C_VEL
LIN {X 0,Y 451.467,Z 734.499,A -85,B 0,C 180,E1 -16733.038,E2 -16733.038} C_VEL
LIN {X 0,Y 450.877,Z 745.305,A -85,B 0,C 180,E1 -16733.393,E2 -16733.393} C_VEL
LIN {X 0,Y 450.225,Z 755.737,A -85,B 0,C 180,E1 -16733.86,E2 -16733.86} C_VEL
LIN {X 0,Y 449.549,Z 765.4,A -85,B 0,C 180,E1 -16734.411,E2 -16734.411} C_VEL
LIN {X 0,Y 448.899,Z 773.454,A -85,B 0,C 180,E1 -16734.964,E2 -16734.964} C_VEL
LIN {X 0,Y 448.018,Z 782.891,A -85,B 0,C 180,E1 -16735.741,E2 -16735.741} C_VEL
LIN {X 0,Y 447.07,Z 791.906,A -85,B 0,C 180,E1 -16736.631,E2 -16736.631} C_VEL
LIN {X 0,Y 446.143,Z 799.592,A -85,B 0,C 180,E1 -16737.525,E2 -16737.525} C_VEL
LIN {X 0,Y 445.287,Z 806.212,A -85,B 0,C 180,E1 -16738.422,E2 -16738.422} C_VEL
LIN {X 0,Y 444.295,Z 813.175,A -85,B 0,C 180,E1 -16739.548,E2 -16739.548} C_VEL
LIN {X 0,Y 443.449,Z 819.941,A -85,B 0,C 180,E1 -16740.905,E2 -16740.905} C_VEL
LIN {X 0,Y 442.947,Z 823.794,A -85,B 0,C 180,E1 -16741.812,E2 -16741.812} C_VEL
LIN {X 0,Y 442.409,Z 828.402,A -85,B 0,C 180,E1 -16743.176,E2 -16743.176} C_VEL
LIN {X 0,Y 442.066,Z 831.889,A -85,B 0,C 180,E1 -16744.544,E2 -16744.544} C_VEL
LIN {X 0,Y 441.617,Z 834.87,A -85,B 0,C 180,E1 -16746.374,E2 -16746.374} C_VEL
LIN {X 0,Y 441.44,Z 835.834,A -85,B 0,C 180,E1 -16747.292,E2 -16747.292} C_VEL
LIN {X 0,Y 441.322,Z 836.218,A -85,B 0,C 180,E1 -16749.132,E2 -16749.132} C_VEL
LIN {X 0,Y 441.376,Z 835.665,A -85,B 0,C 180,E1 -16750.29,E2 -16750.29} C_VEL
LIN {X 0,Y 441.291,Z 833.591,A -85,B 0,C 180,E1 -16751.908,E2 -16751.908} C_VEL
LIN {X 0,Y 441.417,Z 830.711,A -85,B 0,C 180,E1 -16753.302,E2 -16753.302} C_VEL
LIN {X 0,Y 441.642,Z 826.687,A -85,B 0,C 180,E1 -16754.7,E2 -16754.7} C_VEL
LIN {X 0,Y 441.783,Z 822.396,A -85,B 0,C 180,E1 -16755.872,E2 -16755.872} C_VEL
LIN {X 0,Y 442.078,Z 815.859,A -85,B 0,C 180,E1 -16757.282,E2 -16757.282} C_VEL
LIN {X 0,Y 442.396,Z 809.155,A -85,B 0,C 180,E1 -16758.461,E2 -16758.461} C_VEL
LIN {X 0,Y 442.75,Z 802.832,A -85,B 0,C 180,E1 -16759.404,E2 -16759.404} C_VEL
LIN {X 0,Y 443.211,Z 794.315,A -85,B 0,C 180,E1 -16760.466,E2 -16760.466} C_VEL
LIN {X 0,Y 443.657,Z 785.329,A -85,B 0,C 180,E1 -16761.401,E2 -16761.401} C_VEL
LIN {X 0,Y 444.198,Z 775.617,A -85,B 0,C 180,E1 -16762.237,E2 -16762.237} C_VEL
LIN {X 0,Y 444.668,Z 765.604,A -85,B 0,C 180,E1 -16762.946,E2 -16762.946} C_VEL
LIN {X 0,Y 445.121,Z 755.273,A -85,B 0,C 180,E1 -16763.534,E2 -16763.534} C_VEL
LIN {X 0,Y 445.392,Z 744.554,A -85,B 0,C 180,E1 -16764.011,E2 -16764.011} C_VEL
LIN {X 0,Y 445.718,Z 734.23,A -85,B 0,C 180,E1 -16764.351,E2 -16764.351} C_VEL
LIN {X 0,Y 446.292,Z 710.579,A -85,B 0,C 180,E1 -16764.86,E2 -16764.86} C_VEL
LIN {X 0,Y 447.432,Z 651.139,A -85,B 0,C 180,E1 -16766.074,E2 -16766.074} C_VEL
LIN {X 0,Y 444.142,Z 625.597,A -85,B 0,C 180,E1 -16766.695,E2 -16766.695} C_VEL
LIN {X 0,Y 445.007,Z 612.749,A -85,B 0,C 180,E1 -16769.619,E2 -16769.619} C_VEL
LIN {X 0,Y 444.598,Z 607.75,A -85,B 0,C 180,E1 -16770.798,E2 -16770.798} C_VEL
LIN {X 0,Y 443.584,Z 602.164,A -85,B 0,C 180,E1 -16772.173,E2 -16772.173} C_VEL
LIN {X 0,Y 443.501,Z 602.173,A -85,B 0,C 180,E1 -16775.757,E2 -16775.757} C_VEL
LIN {X 0,Y 443.515,Z 602.168,A -85,B 0,C 180,E1 -16779.298,E2 -16779.298} C_VEL
LIN {X 0,Y 443.511,Z 602.168,A -85,B 0,C 180,E1 -16782.773,E2 -16782.773} C_VEL
LIN {X 0,Y 443.517,Z 602.175,A -85,B 0,C 180,E1 -16785.981,E2 -16785.981} C_VEL
LIN {X 0,Y 443.512,Z 602.168,A -85,B 0,C 180,E1 -16789.294,E2 -16789.294} C_VEL
LIN {X 0,Y 443.494,Z 602.175,A -85,B 0,C 180,E1 -16792.155,E2 -16792.155} C_VEL
LIN {X 0,Y 443.525,Z 602.167,A -85,B 0,C 180,E1 -16795.351,E2 -16795.351} C_VEL
LIN {X 0,Y 443.533,Z 602.166,A -85,B 0,C 180,E1 -16798.59,E2 -16798.59} C_VEL
LIN {X 0,Y 443.52,Z 602.171,A -85,B 0,C 180,E1 -16801.719,E2 -16801.719} C_VEL
LIN {X 0,Y 443.489,Z 602.171,A -85,B 0,C 180,E1 -16804.758,E2 -16804.758} C_VEL
LIN {X 0,Y 443.507,Z 602.172,A -85,B 0,C 180,E1 -16807.726,E2 -16807.726} C_VEL
LIN {X 0,Y 443.556,Z 602.163,A -85,B 0,C 180,E1 -16810.632,E2 -16810.632} C_VEL
LIN {X 0,Y 443.672,Z 602.15,A -85,B 0,C 180,E1 -16814.432,E2 -16814.432} C_VEL
LIN {X 0,Y 443.681,Z 602.152,A -85,B 0,C 180,E1 -16818.178,E2 -16818.178} C_VEL
LIN {X 0,Y 443.725,Z 602.147,A -85,B 0,C 180,E1 -16821.832,E2 -16821.832} C_VEL
LIN {X 0,Y 443.777,Z 602.136,A -85,B 0,C 180,E1 -16824.566,E2 -16824.566} C_VEL
LIN {X 0,Y 443.794,Z 602.135,A -85,B 0,C 180,E1 -16826.38,E2 -16826.38} C_VEL
LIN {X 0,Y 443.856,Z 602.133,A -85,B 0,C 180,E1 -16830,E2 -16830} C_VEL
LIN {X 0,Y 443.843,Z 602.128,A -85,B 0,C 180,E1 -16834.526,E2 -16834.526} C_VEL
LIN {X 0,Y 443.744,Z 602.139,A -85,B 0,C 180,E1 -16837.254,E2 -16837.254} C_VEL
LIN {X 0,Y 443.661,Z 602.149,A -85,B 0,C 180,E1 -16840.921,E2 -16840.921} C_VEL
LIN {X 0,Y 443.61,Z 602.159,A -85,B 0,C 180,E1 -16843.7,E2 -16843.7} C_VEL
LIN {X 0,Y 443.643,Z 602.154,A -85,B 0,C 180,E1 -16845.617,E2 -16845.617} C_VEL
LIN {X 0,Y 443.555,Z 602.163,A -85,B 0,C 180,E1 -16849.367,E2 -16849.367} C_VEL
LIN {X 0,Y 443.506,Z 602.172,A -85,B 0,C 180,E1 -16852.274,E2 -16852.274} C_VEL
LIN {X 0,Y 443.488,Z 602.171,A -85,B 0,C 180,E1 -16855.242,E2 -16855.242} C_VEL
LIN {X 0,Y 443.52,Z 602.171,A -85,B 0,C 180,E1 -16858.28,E2 -16858.28} C_VEL
LIN {X 0,Y 443.545,Z 602.165,A -85,B 0,C 180,E1 -16861.487,E2 -16861.487} C_VEL
LIN {X 0,Y 443.564,Z 602.161,A -85,B 0,C 180,E1 -16864.801,E2 -16864.801} C_VEL
LIN {X 0,Y 443.548,Z 602.171,A -85,B 0,C 180,E1 -16868.016,E2 -16868.016} C_VEL
LIN {X 0,Y 443.505,Z 602.169,A -85,B 0,C 180,E1 -16870.047,E2 -16870.047} C_VEL
LIN {X 0,Y 442.863,Z 602.253,A -85,B 0,C 180,E1 -16870.805,E2 -16870.805} C_VEL
LIN {X 0,Y 440.021,Z 602.612,A -85,B 0,C 180,E1 -16872.036,E2 -16872.036} C_VEL
LIN {X 0,Y 437.593,Z 602.913,A -85,B 0,C 180,E1 -16873.03,E2 -16873.03} C_VEL
LIN {X 0,Y 436.538,Z 603.041,A -85,B 0,C 180,E1 -16873.797,E2 -16873.797} C_VEL
LIN {X 0,Y 436.447,Z 603.049,A -85,B 0,C 180,E1 -16874.057,E2 -16874.057} C_VEL
LIN {X 0,Y 436.473,Z 603.047,A -85,B 0,C 180,E1 -16877.578,E2 -16877.578} C_VEL
LIN {X 0,Y 436.464,Z 603.048,A -85,B 0,C 180,E1 -16880.382,E2 -16880.382} C_VEL
LIN {X 0,Y 436.49,Z 603.045,A -85,B 0,C 180,E1 -16883.577,E2 -16883.577} C_VEL
LIN {X 0,Y 436.476,Z 603.044,A -85,B 0,C 180,E1 -16886.933,E2 -16886.933} C_VEL
LIN {X 0,Y 436.487,Z 603.048,A -85,B 0,C 180,E1 -16890.168,E2 -16890.168} C_VEL
LIN {X 0,Y 436.481,Z 603.044,A -85,B 0,C 180,E1 -16893.3,E2 -16893.3} C_VEL
LIN {X 0,Y 436.518,Z 603.042,A -85,B 0,C 180,E1 -16896.35,E2 -16896.35} C_VEL
LIN {X 0,Y 436.488,Z 603.043,A -85,B 0,C 180,E1 -16899.327,E2 -16899.327} C_VEL
LIN {X 0,Y 436.499,Z 603.046,A -85,B 0,C 180,E1 -16902.249,E2 -16902.249} C_VEL
LIN {X 0,Y 436.556,Z 603.034,A -85,B 0,C 180,E1 -16905.125,E2 -16905.125} C_VEL
LIN {X 0,Y 436.632,Z 603.031,A -85,B 0,C 180,E1 -16908.114,E2 -16908.114} C_VEL
LIN {X 0,Y 436.692,Z 603.021,A -85,B 0,C 180,E1 -16911.7,E2 -16911.7} C_VEL
LIN {X 0,Y 436.754,Z 603.011,A -85,B 0,C 180,E1 -16914.478,E2 -16914.478} C_VEL
LIN {X 0,Y 436.683,Z 603.018,A -85,B 0,C 180,E1 -16917.242,E2 -16917.242} C_VEL
LIN {X 0,Y 436.811,Z 603.01,A -85,B 0,C 180,E1 -16920,E2 -16920} C_VEL
LIN {X 0,Y 436.75,Z 603.013,A -85,B 0,C 180,E1 -16923.678,E2 -16923.678} C_VEL
LIN {X 0,Y 436.735,Z 603.014,A -85,B 0,C 180,E1 -16926.446,E2 -16926.446} C_VEL
LIN {X 0,Y 436.622,Z 603.026,A -85,B 0,C 180,E1 -16929.232,E2 -16929.232} C_VEL
LIN {X 0,Y 436.629,Z 603.032,A -85,B 0,C 180,E1 -16932.037,E2 -16932.037} C_VEL
LIN {X 0,Y 436.553,Z 603.034,A -85,B 0,C 180,E1 -16934.876,E2 -16934.876} C_VEL
LIN {X 0,Y 436.525,Z 603.038,A -85,B 0,C 180,E1 -16938.79,E2 -16938.79} C_VEL
LIN {X 0,Y 436.467,Z 603.049,A -85,B 0,C 180,E1 -16941.661,E2 -16941.661} C_VEL
LIN {X 0,Y 436.45,Z 603.048,A -85,B 0,C 180,E1 -16944.662,E2 -16944.662} C_VEL
LIN {X 0,Y 436.494,Z 603.046,A -85,B 0,C 180,E1 -16947.734,E2 -16947.734} C_VEL
LIN {X 0,Y 436.424,Z 603.05,A -85,B 0,C 180,E1 -16950.903,E2 -16950.903} C_VEL
LIN {X 0,Y 436.43,Z 603.055,A -85,B 0,C 180,E1 -16954.176,E2 -16954.176} C_VEL
LIN {X 0,Y 436.443,Z 603.051,A -85,B 0,C 180,E1 -16957.579,E2 -16957.579} C_VEL
LIN {X 0,Y 436.42,Z 603.051,A -85,B 0,C 180,E1 -16961.151,E2 -16961.151} C_VEL
LIN {X 0,Y 436.446,Z 603.052,A -85,B 0,C 180,E1 -16963.764,E2 -16963.764} C_VEL
LIN {X 0,Y 436.445,Z 603.051,A -85,B 0,C 180,E1 -16966.362,E2 -16966.362} C_VEL
LIN {X 0,Y 436.419,Z 603.051,A -85,B 0,C 180,E1 -16968.968,E2 -16968.968} C_VEL
LIN {X 0,Y 436.43,Z 603.052,A -85,B 0,C 180,E1 -16972.42,E2 -16972.42} C_VEL
LIN {X 0,Y 436.412,Z 603.057,A -85,B 0,C 180,E1 -16975.823,E2 -16975.823} C_VEL
LIN {X 0,Y 436.423,Z 603.05,A -85,B 0,C 180,E1 -16979.097,E2 -16979.097} C_VEL
LIN {X 0,Y 436.457,Z 603.051,A -85,B 0,C 180,E1 -16982.264,E2 -16982.264} C_VEL
LIN {X 0,Y 436.546,Z 603.129,A -85,B 0,C 180,E1 -16984.231,E2 -16984.231} C_VEL
LIN {X 0,Y 438.939,Z 616.643,A -85,B 0,C 180,E1 -16987.234,E2 -16987.234} C_VEL
LIN {X 0,Y 438.572,Z 623.591,A -85,B 0,C 180,E1 -16988.695,E2 -16988.695} C_VEL
LIN {X 0,Y 437.116,Z 640.827,A -85,B 0,C 180,E1 -16992.274,E2 -16992.274} C_VEL
LIN {X 0,Y 436.836,Z 645.268,A -85,B 0,C 180,E1 -16993.15,E2 -16993.15} C_VEL
LIN {X 0,Y 439.876,Z 674.751,A -85,B 0,C 180,E1 -16993.855,E2 -16993.855} C_VEL
LIN {X 0,Y 440.171,Z 679.373,A -85,B 0,C 180,E1 -16993.963,E2 -16993.963} C_VEL
LIN {X 0,Y 438.728,Z 751.82,A -85,B 0,C 180,E1 -16995.496,E2 -16995.496} C_VEL
LIN {X 0,Y 438.468,Z 762.014,A -85,B 0,C 180,E1 -16995.812,E2 -16995.812} C_VEL
LIN {X 0,Y 438.085,Z 772.234,A -85,B 0,C 180,E1 -16996.241,E2 -16996.241} C_VEL
LIN {X 0,Y 437.733,Z 780.948,A -85,B 0,C 180,E1 -16996.702,E2 -16996.702} C_VEL
LIN {X 0,Y 437.197,Z 791.395,A -85,B 0,C 180,E1 -16997.392,E2 -16997.392} C_VEL
LIN {X 0,Y 436.625,Z 801.125,A -85,B 0,C 180,E1 -16998.181,E2 -16998.181} C_VEL
LIN {X 0,Y 436.17,Z 810.679,A -85,B 0,C 180,E1 -16999.124,E2 -16999.124} C_VEL
LIN {X 0,Y 435.692,Z 818.551,A -85,B 0,C 180,E1 -17000.048,E2 -17000.048} C_VEL
LIN {X 0,Y 435.302,Z 825.3,A -85,B 0,C 180,E1 -17000.974,E2 -17000.974} C_VEL
LIN {X 0,Y 434.908,Z 832.368,A -85,B 0,C 180,E1 -17002.132,E2 -17002.132} C_VEL
LIN {X 0,Y 434.719,Z 838.274,A -85,B 0,C 180,E1 -17003.292,E2 -17003.292} C_VEL
LIN {X 0,Y 434.552,Z 843.167,A -85,B 0,C 180,E1 -17004.45,E2 -17004.45} C_VEL
LIN {X 0,Y 434.412,Z 847.803,A -85,B 0,C 180,E1 -17005.839,E2 -17005.839} C_VEL
LIN {X 0,Y 434.377,Z 851.287,A -85,B 0,C 180,E1 -17007.227,E2 -17007.227} C_VEL
LIN {X 0,Y 434.36,Z 853.985,A -85,B 0,C 180,E1 -17008.868,E2 -17008.868} C_VEL
LIN {X 0,Y 434.363,Z 855.133,A -85,B 0,C 180,E1 -17010,E2 -17010} C_VEL
LIN {X 0,Y 434.32,Z 855.411,A -85,B 0,C 180,E1 -17011.849,E2 -17011.849} C_VEL
LIN {X 0,Y 434.297,Z 855.022,A -85,B 0,C 180,E1 -17012.774,E2 -17012.774} C_VEL
LIN {X 0,Y 434.45,Z 852.76,A -85,B 0,C 180,E1 -17014.624,E2 -17014.624} C_VEL
LIN {X 0,Y 434.699,Z 849.957,A -85,B 0,C 180,E1 -17016.012,E2 -17016.012} C_VEL
LIN {X 0,Y 435.051,Z 846.089,A -85,B 0,C 180,E1 -17017.401,E2 -17017.401} C_VEL
LIN {X 0,Y 435.639,Z 841.056,A -85,B 0,C 180,E1 -17018.786,E2 -17018.786} C_VEL
LIN {X 0,Y 436.219,Z 835.924,A -85,B 0,C 180,E1 -17019.94,E2 -17019.94} C_VEL
LIN {X 0,Y 437.241,Z 828.287,A -85,B 0,C 180,E1 -17021.317,E2 -17021.317} C_VEL
LIN {X 0,Y 438.263,Z 820.606,A -85,B 0,C 180,E1 -17022.458,E2 -17022.458} C_VEL
LIN {X 0,Y 439.195,Z 813.306,A -85,B 0,C 180,E1 -17023.382,E2 -17023.382} C_VEL
LIN {X 0,Y 440.318,Z 803.722,A -85,B 0,C 180,E1 -17024.392,E2 -17024.392} C_VEL
LIN {X 0,Y 441.281,Z 794.736,A -85,B 0,C 180,E1 -17025.183,E2 -17025.183} C_VEL
LIN {X 0,Y 442.253,Z 785.537,A -85,B 0,C 180,E1 -17025.855,E2 -17025.855} C_VEL
LIN {X 0,Y 443.263,Z 774.093,A -85,B 0,C 180,E1 -17026.525,E2 -17026.525} C_VEL
LIN {X 0,Y 444.169,Z 763.73,A -85,B 0,C 180,E1 -17026.992,E2 -17026.992} C_VEL
LIN {X 0,Y 444.833,Z 753.322,A -85,B 0,C 180,E1 -17027.349,E2 -17027.349} C_VEL
LIN {X 0,Y 445.763,Z 729.748,A -85,B 0,C 180,E1 -17027.902,E2 -17027.902} C_VEL
LIN {X 0,Y 447.575,Z 680.412,A -85,B 0,C 180,E1 -17029.026,E2 -17029.026} C_VEL
LIN {X 0,Y 445.524,Z 666.216,A -85,B 0,C 180,E1 -17029.549,E2 -17029.549} C_VEL
LIN {X 0,Y 442.153,Z 650.417,A -85,B 0,C 180,E1 -17030.221,E2 -17030.221} C_VEL
LIN {X 0,Y 440.391,Z 643.077,A -85,B 0,C 180,E1 -17030.573,E2 -17030.573} C_VEL
LIN {X 0,Y 442.206,Z 631.15,A -85,B 0,C 180,E1 -17033.328,E2 -17033.328} C_VEL
LIN {X 0,Y 441.272,Z 624.104,A -85,B 0,C 180,E1 -17035.207,E2 -17035.207} C_VEL
LIN {X 0,Y 439.729,Z 616.129,A -85,B 0,C 180,E1 -17037.513,E2 -17037.513} C_VEL
LIN {X 0,Y 437.698,Z 607.681,A -85,B 0,C 180,E1 -17040.213,E2 -17040.213} C_VEL
LIN {X 0,Y 436.453,Z 603.051,A -85,B 0,C 180,E1 -17041.852,E2 -17041.852} C_VEL
LIN {X 0,Y 436.471,Z 603.048,A -85,B 0,C 180,E1 -17045.291,E2 -17045.291} C_VEL
LIN {X 0,Y 436.435,Z 603.046,A -85,B 0,C 180,E1 -17048.75,E2 -17048.75} C_VEL
LIN {X 0,Y 436.446,Z 603.046,A -85,B 0,C 180,E1 -17051.148,E2 -17051.148} C_VEL
LIN {X 0,Y 436.459,Z 603.046,A -85,B 0,C 180,E1 -17053.766,E2 -17053.766} C_VEL
LIN {X 0,Y 436.47,Z 603.05,A -85,B 0,C 180,E1 -17056.365,E2 -17056.365} C_VEL
LIN {X 0,Y 436.482,Z 603.046,A -85,B 0,C 180,E1 -17058.959,E2 -17058.959} C_VEL
LIN {X 0,Y 436.458,Z 603.049,A -85,B 0,C 180,E1 -17062.422,E2 -17062.422} C_VEL
LIN {X 0,Y 436.479,Z 603.047,A -85,B 0,C 180,E1 -17065.829,E2 -17065.829} C_VEL
LIN {X 0,Y 436.468,Z 603.05,A -85,B 0,C 180,E1 -17069.1,E2 -17069.1} C_VEL
LIN {X 0,Y 436.502,Z 603.047,A -85,B 0,C 180,E1 -17072.267,E2 -17072.267} C_VEL
LIN {X 0,Y 436.455,Z 603.052,A -85,B 0,C 180,E1 -17075.338,E2 -17075.338} C_VEL
LIN {X 0,Y 436.489,Z 603.052,A -85,B 0,C 180,E1 -17078.341,E2 -17078.341} C_VEL
LIN {X 0,Y 436.549,Z 603.165,A -85,B 0,C 180,E1 -17081.282,E2 -17081.282} C_VEL
LIN {X 0,Y 438.549,Z 611.242,A -85,B 0,C 180,E1 -17084.245,E2 -17084.245} C_VEL
LIN {X 0,Y 440.339,Z 620.062,A -85,B 0,C 180,E1 -17087.132,E2 -17087.132} C_VEL
LIN {X 0,Y 441.322,Z 626.304,A -85,B 0,C 180,E1 -17089.02,E2 -17089.02} C_VEL
LIN {X 0,Y 441.306,Z 628.233,A -85,B 0,C 180,E1 -17089.559,E2 -17089.559} C_VEL
LIN {X 0,Y 446.003,Z 645.614,A -85,B 0,C 180,E1 -17090.403,E2 -17090.403} C_VEL
LIN {X 0,Y 448.331,Z 657.315,A -85,B 0,C 180,E1 -17090.884,E2 -17090.884} C_VEL
LIN {X 0,Y 447.601,Z 673.606,A -85,B 0,C 180,E1 -17091.256,E2 -17091.256} C_VEL
LIN {X 0,Y 445.052,Z 734.788,A -85,B 0,C 180,E1 -17092.657,E2 -17092.657} C_VEL
LIN {X 0,Y 444.446,Z 745.432,A -85,B 0,C 180,E1 -17093.012,E2 -17093.012} C_VEL
LIN {X 0,Y 443.739,Z 755.903,A -85,B 0,C 180,E1 -17093.485,E2 -17093.485} C_VEL
LIN {X 0,Y 443.089,Z 764.708,A -85,B 0,C 180,E1 -17093.988,E2 -17093.988} C_VEL
LIN {X 0,Y 442.276,Z 774.357,A -85,B 0,C 180,E1 -17094.661,E2 -17094.661} C_VEL
LIN {X 0,Y 441.491,Z 782.484,A -85,B 0,C 180,E1 -17095.336,E2 -17095.336} C_VEL
LIN {X 0,Y 440.467,Z 791.592,A -85,B 0,C 180,E1 -17096.239,E2 -17096.239} C_VEL
LIN {X 0,Y 439.377,Z 800.163,A -85,B 0,C 180,E1 -17097.258,E2 -17097.258} C_VEL
LIN {X 0,Y 438.468,Z 806.691,A -85,B 0,C 180,E1 -17098.169,E2 -17098.169} C_VEL
LIN {X 0,Y 437.419,Z 813.586,A -85,B 0,C 180,E1 -17099.312,E2 -17099.312} C_VEL
LIN {X 0,Y 436.683,Z 819.35,A -85,B 0,C 180,E1 -17100.459,E2 -17100.459} C_VEL
LIN {X 0,Y 435.857,Z 824.946,A -85,B 0,C 180,E1 -17101.842,E2 -17101.842} C_VEL
LIN {X 0,Y 435.424,Z 828.039,A -85,B 0,C 180,E1 -17102.766,E2 -17102.766} C_VEL
LIN {X 0,Y 434.954,Z 832.6,A -85,B 0,C 180,E1 -17104.618,E2 -17104.618} C_VEL
LIN {X 0,Y 434.718,Z 834.246,A -85,B 0,C 180,E1 -17105.547,E2 -17105.547} C_VEL
LIN {X 0,Y 434.326,Z 836.156,A -85,B 0,C 180,E1 -17107.412,E2 -17107.412} C_VEL
LIN {X 0,Y 434.249,Z 836.45,A -85,B 0,C 180,E1 -17108.347,E2 -17108.347} C_VEL
LIN {X 0,Y 434.287,Z 835.698,A -85,B 0,C 180,E1 -17110.311,E2 -17110.311} C_VEL
LIN {X 0,Y 434.202,Z 833.235,A -85,B 0,C 180,E1 -17112.105,E2 -17112.105} C_VEL
LIN {X 0,Y 434.29,Z 831.378,A -85,B 0,C 180,E1 -17113.049,E2 -17113.049} C_VEL
LIN {X 0,Y 434.571,Z 826.57,A -85,B 0,C 180,E1 -17114.741,E2 -17114.741} C_VEL
LIN {X 0,Y 434.764,Z 821.322,A -85,B 0,C 180,E1 -17116.135,E2 -17116.135} C_VEL
LIN {X 0,Y 435.007,Z 815.753,A -85,B 0,C 180,E1 -17117.33,E2 -17117.33} C_VEL
LIN {X 0,Y 435.303,Z 809.512,A -85,B 0,C 180,E1 -17118.445,E2 -17118.445} C_VEL
LIN {X 0,Y 435.691,Z 802.584,A -85,B 0,C 180,E1 -17119.486,E2 -17119.486} C_VEL
LIN {X 0,Y 436.152,Z 793.975,A -85,B 0,C 180,E1 -17120.567,E2 -17120.567} C_VEL
LIN {X 0,Y 436.583,Z 785.273,A -85,B 0,C 180,E1 -17121.48,E2 -17121.48} C_VEL
LIN {X 0,Y 437.081,Z 776.596,A -85,B 0,C 180,E1 -17122.247,E2 -17122.247} C_VEL
LIN {X 0,Y 437.573,Z 766.78,A -85,B 0,C 180,E1 -17122.965,E2 -17122.965} C_VEL
LIN {X 0,Y 438.017,Z 756.71,A -85,B 0,C 180,E1 -17123.564,E2 -17123.564} C_VEL
LIN {X 0,Y 438.277,Z 745.574,A -85,B 0,C 180,E1 -17124.081,E2 -17124.081} C_VEL
LIN {X 0,Y 438.662,Z 734.462,A -85,B 0,C 180,E1 -17124.457,E2 -17124.457} C_VEL
LIN {X 0,Y 439.238,Z 712.804,A -85,B 0,C 180,E1 -17124.935,E2 -17124.935} C_VEL
LIN {X 0,Y 440.39,Z 651.537,A -85,B 0,C 180,E1 -17126.222,E2 -17126.222} C_VEL
LIN {X 0,Y 437.118,Z 625.714,A -85,B 0,C 180,E1 -17126.867,E2 -17126.867} C_VEL
LIN {X 0,Y 437.967,Z 613.368,A -85,B 0,C 180,E1 -17129.721,E2 -17129.721} C_VEL
LIN {X 0,Y 437.59,Z 608.817,A -85,B 0,C 180,E1 -17130.811,E2 -17130.811} C_VEL
LIN {X 0,Y 436.561,Z 603.038,A -85,B 0,C 180,E1 -17132.241,E2 -17132.241} C_VEL
LIN {X 0,Y 436.475,Z 603.045,A -85,B 0,C 180,E1 -17135.29,E2 -17135.29} C_VEL
LIN {X 0,Y 436.466,Z 603.046,A -85,B 0,C 180,E1 -17138.746,E2 -17138.746} C_VEL
LIN {X 0,Y 436.477,Z 603.044,A -85,B 0,C 180,E1 -17141.143,E2 -17141.143} C_VEL
LIN {X 0,Y 436.467,Z 603.05,A -85,B 0,C 180,E1 -17143.766,E2 -17143.766} C_VEL
LIN {X 0,Y 436.467,Z 603.048,A -85,B 0,C 180,E1 -17146.364,E2 -17146.364} C_VEL
LIN {X 0,Y 436.479,Z 603.043,A -85,B 0,C 180,E1 -17148.958,E2 -17148.958} C_VEL
LIN {X 0,Y 436.454,Z 603.049,A -85,B 0,C 180,E1 -17152.421,E2 -17152.421} C_VEL
LIN {X 0,Y 436.473,Z 603.05,A -85,B 0,C 180,E1 -17155.828,E2 -17155.828} C_VEL
LIN {X 0,Y 436.462,Z 603.046,A -85,B 0,C 180,E1 -17159.1,E2 -17159.1} C_VEL
LIN {X 0,Y 436.494,Z 603.046,A -85,B 0,C 180,E1 -17162.266,E2 -17162.266} C_VEL
LIN {X 0,Y 436.449,Z 603.048,A -85,B 0,C 180,E1 -17165.338,E2 -17165.338} C_VEL
LIN {X 0,Y 436.483,Z 603.046,A -85,B 0,C 180,E1 -17168.34,E2 -17168.34} C_VEL
LIN {X 0,Y 436.529,Z 603.038,A -85,B 0,C 180,E1 -17171.282,E2 -17171.282} C_VEL
LIN {X 0,Y 436.603,Z 603.028,A -85,B 0,C 180,E1 -17175.126,E2 -17175.126} C_VEL
LIN {X 0,Y 436.63,Z 603.025,A -85,B 0,C 180,E1 -17178.901,E2 -17178.901} C_VEL
LIN {X 0,Y 436.691,Z 603.018,A -85,B 0,C 180,E1 -17182.627,E2 -17182.627} C_VEL
LIN {X 0,Y 436.814,Z 603.003,A -85,B 0,C 180,E1 -17185.401,E2 -17185.401} C_VEL
LIN {X 0,Y 436.698,Z 603.016,A -85,B 0,C 180,E1 -17189.081,E2 -17189.081} C_VEL
LIN {X 0,Y 436.698,Z 603.016,A -85,B 0,C 180,E1 -17190.919,E2 -17190.919} C_VEL
LIN {X 0,Y 436.814,Z 603.003,A -85,B 0,C 180,E1 -17194.599,E2 -17194.599} C_VEL
LIN {X 0,Y 436.691,Z 603.018,A -85,B 0,C 180,E1 -17197.372,E2 -17197.372} C_VEL
LIN {X 0,Y 436.629,Z 603.025,A -85,B 0,C 180,E1 -17201.099,E2 -17201.099} C_VEL
LIN {X 0,Y 436.603,Z 603.028,A -85,B 0,C 180,E1 -17204.874,E2 -17204.874} C_VEL
LIN {X 0,Y 436.529,Z 603.038,A -85,B 0,C 180,E1 -17208.718,E2 -17208.718} C_VEL
LIN {X 0,Y 436.482,Z 603.047,A -85,B 0,C 180,E1 -17211.659,E2 -17211.659} C_VEL
LIN {X 0,Y 436.448,Z 603.048,A -85,B 0,C 180,E1 -17214.662,E2 -17214.662} C_VEL
LIN {X 0,Y 436.493,Z 603.046,A -85,B 0,C 180,E1 -17217.734,E2 -17217.734} C_VEL
LIN {X 0,Y 436.475,Z 603.044,A -85,B 0,C 180,E1 -17220.899,E2 -17220.899} C_VEL
LIN {X 0,Y 436.504,Z 603.046,A -85,B 0,C 180,E1 -17224.169,E2 -17224.169} C_VEL
LIN {X 0,Y 436.514,Z 603.042,A -85,B 0,C 180,E1 -17227.572,E2 -17227.572} C_VEL
LIN {X 0,Y 436.475,Z 603.044,A -85,B 0,C 180,E1 -17231.144,E2 -17231.144} C_VEL
LIN {X 0,Y 436.447,Z 603.049,A -85,B 0,C 180,E1 -17234.057,E2 -17234.057} C_VEL
LIN {X 0,Y 435.767,Z 603.133,A -85,B 0,C 180,E1 -17234.828,E2 -17234.828} C_VEL
LIN {X 0,Y 432.921,Z 603.494,A -85,B 0,C 180,E1 -17236.08,E2 -17236.08} C_VEL
LIN {X 0,Y 430.522,Z 603.797,A -85,B 0,C 180,E1 -17237.091,E2 -17237.091} C_VEL
LIN {X 0,Y 429.491,Z 603.923,A -85,B 0,C 180,E1 -17237.872,E2 -17237.872} C_VEL
LIN {X 0,Y 429.405,Z 603.93,A -85,B 0,C 180,E1 -17238.136,E2 -17238.136} C_VEL
LIN {X 0,Y 429.463,Z 603.92,A -85,B 0,C 180,E1 -17241.524,E2 -17241.524} C_VEL
LIN {X 0,Y 429.432,Z 603.922,A -85,B 0,C 180,E1 -17245.189,E2 -17245.189} C_VEL
LIN {X 0,Y 429.412,Z 603.925,A -85,B 0,C 180,E1 -17248.536,E2 -17248.536} C_VEL
LIN {X 0,Y 429.444,Z 603.925,A -85,B 0,C 180,E1 -17251.771,E2 -17251.771} C_VEL
LIN {X 0,Y 429.41,Z 603.924,A -85,B 0,C 180,E1 -17254.906,E2 -17254.906} C_VEL
LIN {X 0,Y 429.468,Z 603.92,A -85,B 0,C 180,E1 -17258.379,E2 -17258.379} C_VEL
LIN {X 0,Y 429.491,Z 603.914,A -85,B 0,C 180,E1 -17261.068,E2 -17261.068} C_VEL
LIN {X 0,Y 429.501,Z 603.913,A -85,B 0,C 180,E1 -17264.875,E2 -17264.875} C_VEL
LIN {X 0,Y 429.585,Z 603.909,A -85,B 0,C 180,E1 -17268.044,E2 -17268.044} C_VEL
LIN {X 0,Y 429.629,Z 603.899,A -85,B 0,C 180,E1 -17271.563,E2 -17271.563} C_VEL
LIN {X 0,Y 429.716,Z 603.889,A -85,B 0,C 180,E1 -17274.388,E2 -17274.388} C_VEL
LIN {X 0,Y 429.712,Z 603.891,A -85,B 0,C 180,E1 -17276.262,E2 -17276.262} C_VEL
LIN {X 0,Y 429.764,Z 603.888,A -85,B 0,C 180,E1 -17280,E2 -17280} C_VEL
LIN {X 0,Y 429.711,Z 603.891,A -85,B 0,C 180,E1 -17283.739,E2 -17283.739} C_VEL
LIN {X 0,Y 429.69,Z 603.891,A -85,B 0,C 180,E1 -17286.552,E2 -17286.552} C_VEL
LIN {X 0,Y 429.581,Z 603.904,A -85,B 0,C 180,E1 -17289.384,E2 -17289.384} C_VEL
LIN {X 0,Y 429.576,Z 603.908,A -85,B 0,C 180,E1 -17292.238,E2 -17292.238} C_VEL
LIN {X 0,Y 429.478,Z 603.921,A -85,B 0,C 180,E1 -17295.795,E2 -17295.795} C_VEL
LIN {X 0,Y 429.452,Z 603.919,A -85,B 0,C 180,E1 -17299.039,E2 -17299.039} C_VEL
LIN {X 0,Y 429.41,Z 603.931,A -85,B 0,C 180,E1 -17302.035,E2 -17302.035} C_VEL
LIN {X 0,Y 429.408,Z 603.924,A -85,B 0,C 180,E1 -17305.094,E2 -17305.094} C_VEL
LIN {X 0,Y 429.454,Z 603.923,A -85,B 0,C 180,E1 -17308.268,E2 -17308.268} C_VEL
LIN {X 0,Y 429.378,Z 603.93,A -85,B 0,C 180,E1 -17311.468,E2 -17311.468} C_VEL
LIN {X 0,Y 429.393,Z 603.926,A -85,B 0,C 180,E1 -17314.816,E2 -17314.816} C_VEL
LIN {X 0,Y 429.4,Z 603.925,A -85,B 0,C 180,E1 -17317.125,E2 -17317.125} C_VEL
LIN {X 0,Y 429.368,Z 603.93,A -85,B 0,C 180,E1 -17320.733,E2 -17320.733} C_VEL
LIN {X 0,Y 429.398,Z 603.932,A -85,B 0,C 180,E1 -17324.132,E2 -17324.132} C_VEL
LIN {X 0,Y 429.372,Z 603.929,A -85,B 0,C 180,E1 -17327.231,E2 -17327.231} C_VEL
LIN {X 0,Y 429.365,Z 603.932,A -85,B 0,C 180,E1 -17330.489,E2 -17330.489} C_VEL
LIN {X 0,Y 429.388,Z 603.927,A -85,B 0,C 180,E1 -17333.065,E2 -17333.065} C_VEL
LIN {X 0,Y 429.366,Z 603.933,A -85,B 0,C 180,E1 -17336.313,E2 -17336.313} C_VEL
LIN {X 0,Y 429.394,Z 603.929,A -85,B 0,C 180,E1 -17339.623,E2 -17339.623} C_VEL
LIN {X 0,Y 429.424,Z 603.922,A -85,B 0,C 180,E1 -17342.825,E2 -17342.825} C_VEL
LIN {X 0,Y 429.508,Z 604.029,A -85,B 0,C 180,E1 -17344.136,E2 -17344.136} C_VEL
LIN {X 0,Y 431.985,Z 618.49,A -85,B 0,C 180,E1 -17347.388,E2 -17347.388} C_VEL
LIN {X 0,Y 430.899,Z 630.984,A -85,B 0,C 180,E1 -17350.04,E2 -17350.04} C_VEL
LIN {X 0,Y 429.779,Z 644.867,A -85,B 0,C 180,E1 -17352.965,E2 -17352.965} C_VEL
LIN {X 0,Y 432.958,Z 676.099,A -85,B 0,C 180,E1 -17353.744,E2 -17353.744} C_VEL
LIN {X 0,Y 433.104,Z 683.881,A -85,B 0,C 180,E1 -17353.92,E2 -17353.92} C_VEL
LIN {X 0,Y 431.711,Z 751.321,A -85,B 0,C 180,E1 -17355.375,E2 -17355.375} C_VEL
LIN {X 0,Y 431.425,Z 761.585,A -85,B 0,C 180,E1 -17355.695,E2 -17355.695} C_VEL
LIN {X 0,Y 431.058,Z 771.863,A -85,B 0,C 180,E1 -17356.133,E2 -17356.133} C_VEL
LIN {X 0,Y 430.612,Z 782.449,A -85,B 0,C 180,E1 -17356.717,E2 -17356.717} C_VEL
LIN {X 0,Y 430.08,Z 792.586,A -85,B 0,C 180,E1 -17357.419,E2 -17357.419} C_VEL
LIN {X 0,Y 429.535,Z 801.225,A -85,B 0,C 180,E1 -17358.139,E2 -17358.139} C_VEL
LIN {X 0,Y 429.202,Z 809.39,A -85,B 0,C 180,E1 -17358.945,E2 -17358.945} C_VEL
LIN {X 0,Y 428.645,Z 817.438,A -85,B 0,C 180,E1 -17359.883,E2 -17359.883} C_VEL
LIN {X 0,Y 428.168,Z 825.805,A -85,B 0,C 180,E1 -17361.06,E2 -17361.06} C_VEL
LIN {X 0,Y 427.818,Z 832.77,A -85,B 0,C 180,E1 -17362.237,E2 -17362.237} C_VEL
LIN {X 0,Y 427.614,Z 838.576,A -85,B 0,C 180,E1 -17363.416,E2 -17363.416} C_VEL
LIN {X 0,Y 427.432,Z 844.176,A -85,B 0,C 180,E1 -17364.829,E2 -17364.829} C_VEL
LIN {X 0,Y 427.343,Z 847.3,A -85,B 0,C 180,E1 -17365.77,E2 -17365.77} C_VEL
LIN {X 0,Y 427.286,Z 850.882,A -85,B 0,C 180,E1 -17367.181,E2 -17367.181} C_VEL
LIN {X 0,Y 427.289,Z 853.906,A -85,B 0,C 180,E1 -17369.061,E2 -17369.061} C_VEL
LIN {X 0,Y 427.271,Z 854.87,A -85,B 0,C 180,E1 -17370,E2 -17370} C_VEL
LIN {X 0,Y 427.246,Z 855.287,A -85,B 0,C 180,E1 -17371.879,E2 -17371.879} C_VEL
LIN {X 0,Y 427.222,Z 854.902,A -85,B 0,C 180,E1 -17372.819,E2 -17372.819} C_VEL
LIN {X 0,Y 427.373,Z 852.814,A -85,B 0,C 180,E1 -17374.701,E2 -17374.701} C_VEL
LIN {X 0,Y 427.648,Z 850.098,A -85,B 0,C 180,E1 -17376.112,E2 -17376.112} C_VEL
LIN {X 0,Y 428.021,Z 846.319,A -85,B 0,C 180,E1 -17377.523,E2 -17377.523} C_VEL
LIN {X 0,Y 428.637,Z 841.377,A -85,B 0,C 180,E1 -17378.931,E2 -17378.931} C_VEL
LIN {X 0,Y 429.449,Z 835.159,A -85,B 0,C 180,E1 -17380.336,E2 -17380.336} C_VEL
LIN {X 0,Y 430.317,Z 828.907,A -85,B 0,C 180,E1 -17381.502,E2 -17381.502} C_VEL
LIN {X 0,Y 431.341,Z 821.757,A -85,B 0,C 180,E1 -17382.614,E2 -17382.614} C_VEL
LIN {X 0,Y 432.582,Z 812.542,A -85,B 0,C 180,E1 -17383.794,E2 -17383.794} C_VEL
LIN {X 0,Y 433.658,Z 803.696,A -85,B 0,C 180,E1 -17384.738,E2 -17384.738} C_VEL
LIN {X 0,Y 434.684,Z 794.727,A -85,B 0,C 180,E1 -17385.539,E2 -17385.539} C_VEL
LIN {X 0,Y 435.709,Z 785.557,A -85,B 0,C 180,E1 -17386.22,E2 -17386.22} C_VEL
LIN {X 0,Y 436.779,Z 774.163,A -85,B 0,C 180,E1 -17386.898,E2 -17386.898} C_VEL
LIN {X 0,Y 437.764,Z 763.201,A -85,B 0,C 180,E1 -17387.398,E2 -17387.398} C_VEL
LIN {X 0,Y 438.461,Z 752.862,A -85,B 0,C 180,E1 -17387.76,E2 -17387.76} C_VEL
LIN {X 0,Y 439.487,Z 728.549,A -85,B 0,C 180,E1 -17388.347,E2 -17388.347} C_VEL
LIN {X 0,Y 441.343,Z 681.337,A -85,B 0,C 180,E1 -17389.451,E2 -17389.451} C_VEL
LIN {X 0,Y 438.978,Z 665.584,A -85,B 0,C 180,E1 -17390.053,E2 -17390.053} C_VEL
LIN {X 0,Y 435.001,Z 647.68,A -85,B 0,C 180,E1 -17390.877,E2 -17390.877} C_VEL
LIN {X 0,Y 433.806,Z 642.898,A -85,B 0,C 180,E1 -17391.115,E2 -17391.115} C_VEL
LIN {X 0,Y 435.406,Z 632.762,A -85,B 0,C 180,E1 -17393.513,E2 -17393.513} C_VEL
LIN {X 0,Y 434.437,Z 625.677,A -85,B 0,C 180,E1 -17395.459,E2 -17395.459} C_VEL
LIN {X 0,Y 432.832,Z 617.199,A -85,B 0,C 180,E1 -17397.989,E2 -17397.989} C_VEL
LIN {X 0,Y 430.665,Z 608.722,A -85,B 0,C 180,E1 -17400.838,E2 -17400.838} C_VEL
LIN {X 0,Y 429.397,Z 603.933,A -85,B 0,C 180,E1 -17402.638,E2 -17402.638} C_VEL
LIN {X 0,Y 429.416,Z 603.925,A -85,B 0,C 180,E1 -17405.96,E2 -17405.96} C_VEL
LIN {X 0,Y 429.387,Z 603.923,A -85,B 0,C 180,E1 -17409.509,E2 -17409.509} C_VEL
LIN {X 0,Y 429.384,Z 603.929,A -85,B 0,C 180,E1 -17412.771,E2 -17412.771} C_VEL
LIN {X 0,Y 429.417,Z 603.928,A -85,B 0,C 180,E1 -17415.866,E2 -17415.866} C_VEL
LIN {X 0,Y 429.441,Z 603.924,A -85,B 0,C 180,E1 -17419.275,E2 -17419.275} C_VEL
LIN {X 0,Y 429.416,Z 603.929,A -85,B 0,C 180,E1 -17421.695,E2 -17421.695} C_VEL
LIN {X 0,Y 429.43,Z 603.928,A -85,B 0,C 180,E1 -17425.188,E2 -17425.188} C_VEL
LIN {X 0,Y 429.418,Z 603.927,A -85,B 0,C 180,E1 -17428.536,E2 -17428.536} C_VEL
LIN {X 0,Y 429.448,Z 603.923,A -85,B 0,C 180,E1 -17431.771,E2 -17431.771} C_VEL
LIN {X 0,Y 429.415,Z 603.93,A -85,B 0,C 180,E1 -17434.906,E2 -17434.906} C_VEL
LIN {X 0,Y 429.472,Z 603.926,A -85,B 0,C 180,E1 -17438.379,E2 -17438.379} C_VEL
LIN {X 0,Y 429.498,Z 604.07,A -85,B 0,C 180,E1 -17440.537,E2 -17440.537} C_VEL
LIN {X 0,Y 431.314,Z 611.405,A -85,B 0,C 180,E1 -17443.366,E2 -17443.366} C_VEL
LIN {X 0,Y 432.972,Z 618.84,A -85,B 0,C 180,E1 -17445.956,E2 -17445.956} C_VEL
LIN {X 0,Y 434.342,Z 626.395,A -85,B 0,C 180,E1 -17448.37,E2 -17448.37} C_VEL
LIN {X 0,Y 434.563,Z 628.623,A -85,B 0,C 180,E1 -17449.008,E2 -17449.008} C_VEL
LIN {X 0,Y 437.663,Z 638.522,A -85,B 0,C 180,E1 -17449.554,E2 -17449.554} C_VEL
LIN {X 0,Y 440.985,Z 652.526,A -85,B 0,C 180,E1 -17450.21,E2 -17450.21} C_VEL
LIN {X 0,Y 442.14,Z 659.335,A -85,B 0,C 180,E1 -17450.479,E2 -17450.479} C_VEL
LIN {X 0,Y 438.738,Z 734.399,A -85,B 0,C 180,E1 -17452.233,E2 -17452.233} C_VEL
LIN {X 0,Y 438.093,Z 744.513,A -85,B 0,C 180,E1 -17452.568,E2 -17452.568} C_VEL
LIN {X 0,Y 437.399,Z 755.014,A -85,B 0,C 180,E1 -17453.043,E2 -17453.043} C_VEL
LIN {X 0,Y 436.69,Z 763.992,A -85,B 0,C 180,E1 -17453.553,E2 -17453.553} C_VEL
LIN {X 0,Y 435.778,Z 773.843,A -85,B 0,C 180,E1 -17454.234,E2 -17454.234} C_VEL
LIN {X 0,Y 434.84,Z 783.279,A -85,B 0,C 180,E1 -17455.033,E2 -17455.033} C_VEL
LIN {X 0,Y 433.769,Z 792.299,A -85,B 0,C 180,E1 -17455.949,E2 -17455.949} C_VEL
LIN {X 0,Y 432.905,Z 799.097,A -85,B 0,C 180,E1 -17456.753,E2 -17456.753} C_VEL
LIN {X 0,Y 431.674,Z 807.268,A -85,B 0,C 180,E1 -17457.907,E2 -17457.907} C_VEL
LIN {X 0,Y 430.582,Z 814.095,A -85,B 0,C 180,E1 -17459.068,E2 -17459.068} C_VEL
LIN {X 0,Y 429.908,Z 818.786,A -85,B 0,C 180,E1 -17460,E2 -17460} C_VEL
LIN {X 0,Y 429.077,Z 824.52,A -85,B 0,C 180,E1 -17461.403,E2 -17461.403} C_VEL
LIN {X 0,Y 428.36,Z 829.054,A -85,B 0,C 180,E1 -17462.811,E2 -17462.811} C_VEL
LIN {X 0,Y 428.148,Z 831.389,A -85,B 0,C 180,E1 -17463.752,E2 -17463.752} C_VEL
LIN {X 0,Y 427.607,Z 834.862,A -85,B 0,C 180,E1 -17465.64,E2 -17465.64} C_VEL
LIN {X 0,Y 427.212,Z 836.428,A -85,B 0,C 180,E1 -17467.537,E2 -17467.537} C_VEL
LIN {X 0,Y 427.162,Z 836.69,A -85,B 0,C 180,E1 -17468.486,E2 -17468.486} C_VEL
LIN {X 0,Y 427.191,Z 835.641,A -85,B 0,C 180,E1 -17470.39,E2 -17470.39} C_VEL
LIN {X 0,Y 427.099,Z 834.56,A -85,B 0,C 180,E1 -17471.35,E2 -17471.35} C_VEL
LIN {X 0,Y 427.168,Z 831.962,A -85,B 0,C 180,E1 -17472.789,E2 -17472.789} C_VEL
LIN {X 0,Y 427.387,Z 828.264,A -85,B 0,C 180,E1 -17474.231,E2 -17474.231} C_VEL
LIN {X 0,Y 427.615,Z 822.291,A -85,B 0,C 180,E1 -17475.924,E2 -17475.924} C_VEL
LIN {X 0,Y 427.883,Z 816.903,A -85,B 0,C 180,E1 -17477.137,E2 -17477.137} C_VEL
LIN {X 0,Y 428.205,Z 809.896,A -85,B 0,C 180,E1 -17478.423,E2 -17478.423} C_VEL
LIN {X 0,Y 428.62,Z 802.329,A -85,B 0,C 180,E1 -17479.573,E2 -17479.573} C_VEL
LIN {X 0,Y 429.063,Z 794.724,A -85,B 0,C 180,E1 -17480.547,E2 -17480.547} C_VEL
LIN {X 0,Y 429.5,Z 785.405,A -85,B 0,C 180,E1 -17481.544,E2 -17481.544} C_VEL
LIN {X 0,Y 430.06,Z 776.024,A -85,B 0,C 180,E1 -17482.377,E2 -17482.377} C_VEL
LIN {X 0,Y 430.559,Z 766.037,A -85,B 0,C 180,E1 -17483.108,E2 -17483.108} C_VEL
LIN {X 0,Y 431.014,Z 755.733,A -85,B 0,C 180,E1 -17483.716,E2 -17483.716} C_VEL
LIN {X 0,Y 431.262,Z 745.401,A -85,B 0,C 180,E1 -17484.197,E2 -17484.197} C_VEL
LIN {X 0,Y 431.625,Z 734.239,A -85,B 0,C 180,E1 -17484.578,E2 -17484.578} C_VEL
LIN {X 0,Y 432.231,Z 711.918,A -85,B 0,C 180,E1 -17485.079,E2 -17485.079} C_VEL
LIN {X 0,Y 433.389,Z 652.059,A -85,B 0,C 180,E1 -17486.362,E2 -17486.362} C_VEL
LIN {X 0,Y 430.101,Z 625.915,A -85,B 0,C 180,E1 -17487.027,E2 -17487.027} C_VEL
LIN {X 0,Y 430.96,Z 613.311,A -85,B 0,C 180,E1 -17489.985,E2 -17489.985} C_VEL
LIN {X 0,Y 429.889,Z 606.227,A -85,B 0,C 180,E1 -17491.723,E2 -17491.723} C_VEL
LIN {X 0,Y 429.521,Z 603.914,A -85,B 0,C 180,E1 -17492.331,E2 -17492.331} C_VEL
LIN {X 0,Y 429.417,Z 603.931,A -85,B 0,C 180,E1 -17495.959,E2 -17495.959} C_VEL
LIN {X 0,Y 429.436,Z 603.923,A -85,B 0,C 180,E1 -17499.502,E2 -17499.502} C_VEL
LIN {X 0,Y 429.432,Z 603.922,A -85,B 0,C 180,E1 -17502.778,E2 -17502.778} C_VEL
LIN {X 0,Y 429.415,Z 603.93,A -85,B 0,C 180,E1 -17505.865,E2 -17505.865} C_VEL
LIN {X 0,Y 429.438,Z 603.921,A -85,B 0,C 180,E1 -17509.275,E2 -17509.275} C_VEL
LIN {X 0,Y 429.412,Z 603.928,A -85,B 0,C 180,E1 -17511.695,E2 -17511.695} C_VEL
LIN {X 0,Y 429.43,Z 603.922,A -85,B 0,C 180,E1 -17515.188,E2 -17515.188} C_VEL
LIN {X 0,Y 429.412,Z 603.926,A -85,B 0,C 180,E1 -17518.535,E2 -17518.535} C_VEL
LIN {X 0,Y 429.443,Z 603.925,A -85,B 0,C 180,E1 -17521.77,E2 -17521.77} C_VEL
LIN {X 0,Y 429.409,Z 603.924,A -85,B 0,C 180,E1 -17524.906,E2 -17524.906} C_VEL
LIN {X 0,Y 429.466,Z 603.92,A -85,B 0,C 180,E1 -17528.379,E2 -17528.379} C_VEL
LIN {X 0,Y 429.489,Z 603.914,A -85,B 0,C 180,E1 -17531.067,E2 -17531.067} C_VEL
LIN {X 0,Y 429.546,Z 603.907,A -85,B 0,C 180,E1 -17534.876,E2 -17534.876} C_VEL
LIN {X 0,Y 429.603,Z 603.901,A -85,B 0,C 180,E1 -17538.717,E2 -17538.717} C_VEL
LIN {X 0,Y 429.642,Z 603.897,A -85,B 0,C 180,E1 -17542.506,E2 -17542.506} C_VEL
LIN {X 0,Y 429.785,Z 603.878,A -85,B 0,C 180,E1 -17545.326,E2 -17545.326} C_VEL
LIN {X 0,Y 429.65,Z 603.894,A -85,B 0,C 180,E1 -17549.066,E2 -17549.066} C_VEL
LIN {X 0,Y 429.649,Z 603.894,A -85,B 0,C 180,E1 -17550.934,E2 -17550.934} C_VEL
LIN {X 0,Y 429.785,Z 603.878,A -85,B 0,C 180,E1 -17554.674,E2 -17554.674} C_VEL
LIN {X 0,Y 429.642,Z 603.897,A -85,B 0,C 180,E1 -17557.494,E2 -17557.494} C_VEL
LIN {X 0,Y 429.603,Z 603.901,A -85,B 0,C 180,E1 -17561.283,E2 -17561.283} C_VEL
LIN {X 0,Y 429.545,Z 603.907,A -85,B 0,C 180,E1 -17565.124,E2 -17565.124} C_VEL
LIN {X 0,Y 429.489,Z 603.914,A -85,B 0,C 180,E1 -17568.933,E2 -17568.933} C_VEL
LIN {X 0,Y 429.441,Z 603.928,A -85,B 0,C 180,E1 -17572.033,E2 -17572.033} C_VEL
LIN {X 0,Y 429.407,Z 603.924,A -85,B 0,C 180,E1 -17575.094,E2 -17575.094} C_VEL
LIN {X 0,Y 429.45,Z 603.923,A -85,B 0,C 180,E1 -17578.268,E2 -17578.268} C_VEL
LIN {X 0,Y 429.462,Z 603.925,A -85,B 0,C 180,E1 -17581.994,E2 -17581.994} C_VEL
LIN {X 0,Y 429.452,Z 603.919,A -85,B 0,C 180,E1 -17584.81,E2 -17584.81} C_VEL
LIN {X 0,Y 429.473,Z 603.916,A -85,B 0,C 180,E1 -17587.117,E2 -17587.117} C_VEL
LIN {X 0,Y 429.439,Z 603.928,A -85,B 0,C 180,E1 -17589.951,E2 -17589.951} C_VEL
LIN {X 0,Y 429.426,Z 603.922,A -85,B 0,C 180,E1 -17593.241,E2 -17593.241} C_VEL
LIN {X 0,Y 429.426,Z 603.922,A -85,B 0,C 180,E1 -17596.76,E2 -17596.76} C_VEL
LIN {X 0,Y 429.405,Z 603.93,A -85,B 0,C 180,E1 -17598.136,E2 -17598.136} C_VEL
LIN {X 0,Y 428.743,Z 604.008,A -85,B 0,C 180,E1 -17598.919,E2 -17598.919} C_VEL
LIN {X 0,Y 425.921,Z 604.364,A -85,B 0,C 180,E1 -17600.192,E2 -17600.192} C_VEL
LIN {X 0,Y 423.524,Z 604.666,A -85,B 0,C 180,E1 -17601.22,E2 -17601.22} C_VEL
LIN {X 0,Y 422.482,Z 604.795,A -85,B 0,C 180,E1 -17602.013,E2 -17602.013} C_VEL
LIN {X 0,Y 422.39,Z 604.803,A -85,B 0,C 180,E1 -17602.282,E2 -17602.282} C_VEL
LIN {X 0,Y 422.416,Z 604.797,A -85,B 0,C 180,E1 -17604.524,E2 -17604.524} C_VEL
LIN {X 0,Y 422.381,Z 604.807,A -85,B 0,C 180,E1 -17607.95,E2 -17607.95} C_VEL
LIN {X 0,Y 422.404,Z 604.799,A -85,B 0,C 180,E1 -17611.505,E2 -17611.505} C_VEL
LIN {X 0,Y 422.389,Z 604.801,A -85,B 0,C 180,E1 -17614.46,E2 -17614.46} C_VEL
LIN {X 0,Y 422.4,Z 604.8,A -85,B 0,C 180,E1 -17617.58,E2 -17617.58} C_VEL
LIN {X 0,Y 422.448,Z 604.791,A -85,B 0,C 180,E1 -17620.925,E2 -17620.925} C_VEL
LIN {X 0,Y 422.465,Z 604.79,A -85,B 0,C 180,E1 -17624.617,E2 -17624.617} C_VEL
LIN {X 0,Y 422.562,Z 604.779,A -85,B 0,C 180,E1 -17628.527,E2 -17628.527} C_VEL
LIN {X 0,Y 422.636,Z 604.771,A -85,B 0,C 180,E1 -17632.381,E2 -17632.381} C_VEL
LIN {X 0,Y 422.741,Z 604.755,A -85,B 0,C 180,E1 -17635.248,E2 -17635.248} C_VEL
LIN {X 0,Y 422.551,Z 604.785,A -85,B 0,C 180,E1 -17638.1,E2 -17638.1} C_VEL
LIN {X 0,Y 422.718,Z 604.766,A -85,B 0,C 180,E1 -17640,E2 -17640} C_VEL
LIN {X 0,Y 422.675,Z 604.768,A -85,B 0,C 180,E1 -17643.801,E2 -17643.801} C_VEL
LIN {X 0,Y 422.639,Z 604.768,A -85,B 0,C 180,E1 -17646.662,E2 -17646.662} C_VEL
LIN {X 0,Y 422.525,Z 604.784,A -85,B 0,C 180,E1 -17649.543,E2 -17649.543} C_VEL
LIN {X 0,Y 422.517,Z 604.785,A -85,B 0,C 180,E1 -17652.446,E2 -17652.446} C_VEL
LIN {X 0,Y 422.419,Z 604.801,A -85,B 0,C 180,E1 -17655.901,E2 -17655.901} C_VEL
LIN {X 0,Y 422.381,Z 604.801,A -85,B 0,C 180,E1 -17659.37,E2 -17659.37} C_VEL
LIN {X 0,Y 422.381,Z 604.802,A -85,B 0,C 180,E1 -17662.421,E2 -17662.421} C_VEL
LIN {X 0,Y 422.387,Z 604.801,A -85,B 0,C 180,E1 -17665.541,E2 -17665.541} C_VEL
LIN {X 0,Y 422.39,Z 604.799,A -85,B 0,C 180,E1 -17668.745,E2 -17668.745} C_VEL
LIN {X 0,Y 422.347,Z 604.811,A -85,B 0,C 180,E1 -17672.053,E2 -17672.053} C_VEL
LIN {X 0,Y 422.378,Z 604.803,A -85,B 0,C 180,E1 -17675.651,E2 -17675.651} C_VEL
LIN {X 0,Y 422.317,Z 604.808,A -85,B 0,C 180,E1 -17679.069,E2 -17679.069} C_VEL
LIN {X 0,Y 422.315,Z 604.812,A -85,B 0,C 180,E1 -17681.724,E2 -17681.724} C_VEL
LIN {X 0,Y 422.359,Z 604.804,A -85,B 0,C 180,E1 -17684.511,E2 -17684.511} C_VEL
LIN {X 0,Y 422.326,Z 604.807,A -85,B 0,C 180,E1 -17687.156,E2 -17687.156} C_VEL
LIN {X 0,Y 422.349,Z 604.808,A -85,B 0,C 180,E1 -17689.719,E2 -17689.719} C_VEL
LIN {X 0,Y 422.332,Z 604.807,A -85,B 0,C 180,E1 -17693.34,E2 -17693.34} C_VEL
LIN {X 0,Y 422.299,Z 604.81,A -85,B 0,C 180,E1 -17696.815,E2 -17696.815} C_VEL
LIN {X 0,Y 422.349,Z 604.809,A -85,B 0,C 180,E1 -17700.163,E2 -17700.163} C_VEL
LIN {X 0,Y 422.413,Z 604.798,A -85,B 0,C 180,E1 -17703.563,E2 -17703.563} C_VEL
LIN {X 0,Y 422.435,Z 604.906,A -85,B 0,C 180,E1 -17704.034,E2 -17704.034} C_VEL
LIN {X 0,Y 424.833,Z 618.224,A -85,B 0,C 180,E1 -17707.089,E2 -17707.089} C_VEL
LIN {X 0,Y 424.654,Z 623.39,A -85,B 0,C 180,E1 -17708.215,E2 -17708.215} C_VEL
LIN {X 0,Y 423.085,Z 640.608,A -85,B 0,C 180,E1 -17711.916,E2 -17711.916} C_VEL
LIN {X 0,Y 422.745,Z 644.791,A -85,B 0,C 180,E1 -17712.809,E2 -17712.809} C_VEL
LIN {X 0,Y 425.984,Z 677.027,A -85,B 0,C 180,E1 -17713.618,E2 -17713.618} C_VEL
LIN {X 0,Y 425.984,Z 689.068,A -85,B 0,C 180,E1 -17713.891,E2 -17713.891} C_VEL
LIN {X 0,Y 424.661,Z 751.878,A -85,B 0,C 180,E1 -17715.279,E2 -17715.279} C_VEL
LIN {X 0,Y 424.367,Z 761.902,A -85,B 0,C 180,E1 -17715.605,E2 -17715.605} C_VEL
LIN {X 0,Y 424.006,Z 771.474,A -85,B 0,C 180,E1 -17716.019,E2 -17716.019} C_VEL
LIN {X 0,Y 423.563,Z 782.106,A -85,B 0,C 180,E1 -17716.614,E2 -17716.614} C_VEL
LIN {X 0,Y 423.029,Z 792.28,A -85,B 0,C 180,E1 -17717.327,E2 -17717.327} C_VEL
LIN {X 0,Y 422.443,Z 801.336,A -85,B 0,C 180,E1 -17718.097,E2 -17718.097} C_VEL
LIN {X 0,Y 422.041,Z 810.167,A -85,B 0,C 180,E1 -17718.997,E2 -17718.997} C_VEL
LIN {X 0,Y 421.539,Z 818.061,A -85,B 0,C 180,E1 -17719.952,E2 -17719.952} C_VEL
LIN {X 0,Y 421.143,Z 824.831,A -85,B 0,C 180,E1 -17720.909,E2 -17720.909} C_VEL
LIN {X 0,Y 420.74,Z 831.92,A -85,B 0,C 180,E1 -17722.106,E2 -17722.106} C_VEL
LIN {X 0,Y 420.534,Z 837.844,A -85,B 0,C 180,E1 -17723.305,E2 -17723.305} C_VEL
LIN {X 0,Y 420.35,Z 843.552,A -85,B 0,C 180,E1 -17724.742,E2 -17724.742} C_VEL
LIN {X 0,Y 420.257,Z 848.005,A -85,B 0,C 180,E1 -17726.178,E2 -17726.178} C_VEL
LIN {X 0,Y 420.217,Z 850.389,A -85,B 0,C 180,E1 -17727.134,E2 -17727.134} C_VEL
LIN {X 0,Y 420.209,Z 853.589,A -85,B 0,C 180,E1 -17729.045,E2 -17729.045} C_VEL
LIN {X 0,Y 420.186,Z 854.562,A -85,B 0,C 180,E1 -17730,E2 -17730} C_VEL
LIN {X 0,Y 420.168,Z 855.163,A -85,B 0,C 180,E1 -17731.911,E2 -17731.911} C_VEL
LIN {X 0,Y 420.145,Z 854.776,A -85,B 0,C 180,E1 -17732.867,E2 -17732.867} C_VEL
LIN {X 0,Y 420.311,Z 852.857,A -85,B 0,C 180,E1 -17734.78,E2 -17734.78} C_VEL
LIN {X 0,Y 420.587,Z 850.218,A -85,B 0,C 180,E1 -17736.215,E2 -17736.215} C_VEL
LIN {X 0,Y 421,Z 846.549,A -85,B 0,C 180,E1 -17737.649,E2 -17737.649} C_VEL
LIN {X 0,Y 421.643,Z 841.76,A -85,B 0,C 180,E1 -17739.08,E2 -17739.08} C_VEL
LIN {X 0,Y 422.503,Z 835.693,A -85,B 0,C 180,E1 -17740.508,E2 -17740.508} C_VEL
LIN {X 0,Y 423.64,Z 828.12,A -85,B 0,C 180,E1 -17741.928,E2 -17741.928} C_VEL
LIN {X 0,Y 424.726,Z 820.233,A -85,B 0,C 180,E1 -17743.143,E2 -17743.143} C_VEL
LIN {X 0,Y 425.915,Z 812.395,A -85,B 0,C 180,E1 -17744.148,E2 -17744.148} C_VEL
LIN {X 0,Y 427.042,Z 803.659,A -85,B 0,C 180,E1 -17745.093,E2 -17745.093} C_VEL
LIN {X 0,Y 428.127,Z 794.775,A -85,B 0,C 180,E1 -17745.905,E2 -17745.905} C_VEL
LIN {X 0,Y 429.35,Z 783.994,A -85,B 0,C 180,E1 -17746.711,E2 -17746.711} C_VEL
LIN {X 0,Y 430.421,Z 773.491,A -85,B 0,C 180,E1 -17747.338,E2 -17747.338} C_VEL
LIN {X 0,Y 431.411,Z 763.213,A -85,B 0,C 180,E1 -17747.816,E2 -17747.816} C_VEL
LIN {X 0,Y 432.157,Z 752.001,A -85,B 0,C 180,E1 -17748.211,E2 -17748.211} C_VEL
LIN {X 0,Y 433.978,Z 711.036,A -85,B 0,C 180,E1 -17749.194,E2 -17749.194} C_VEL
LIN {X 0,Y 435.098,Z 682.04,A -85,B 0,C 180,E1 -17749.898,E2 -17749.898} C_VEL
LIN {X 0,Y 432.946,Z 667.271,A -85,B 0,C 180,E1 -17750.489,E2 -17750.489} C_VEL
LIN {X 0,Y 429.024,Z 649.637,A -85,B 0,C 180,E1 -17751.33,E2 -17751.33} C_VEL
LIN {X 0,Y 427.274,Z 642.7,A -85,B 0,C 180,E1 -17751.695,E2 -17751.695} C_VEL
LIN {X 0,Y 428.607,Z 634.198,A -85,B 0,C 180,E1 -17753.77,E2 -17753.77} C_VEL
LIN {X 0,Y 427.609,Z 627.28,A -85,B 0,C 180,E1 -17755.72,E2 -17755.72} C_VEL
LIN {X 0,Y 425.889,Z 618.343,A -85,B 0,C 180,E1 -17758.487,E2 -17758.487} C_VEL
LIN {X 0,Y 424.176,Z 611.582,A -85,B 0,C 180,E1 -17760.831,E2 -17760.831} C_VEL
LIN {X 0,Y 422.36,Z 604.808,A -85,B 0,C 180,E1 -17763.517,E2 -17763.517} C_VEL
LIN {X 0,Y 422.359,Z 604.803,A -85,B 0,C 180,E1 -17766.658,E2 -17766.658} C_VEL
LIN {X 0,Y 422.373,Z 604.796,A -85,B 0,C 180,E1 -17770.298,E2 -17770.298} C_VEL
LIN {X 0,Y 422.382,Z 604.803,A -85,B 0,C 180,E1 -17774.147,E2 -17774.147} C_VEL
LIN {X 0,Y 422.388,Z 604.802,A -85,B 0,C 180,E1 -17777.164,E2 -17777.164} C_VEL
LIN {X 0,Y 422.405,Z 604.803,A -85,B 0,C 180,E1 -17779.711,E2 -17779.711} C_VEL
LIN {X 0,Y 422.362,Z 604.808,A -85,B 0,C 180,E1 -17783.343,E2 -17783.343} C_VEL
LIN {X 0,Y 422.388,Z 604.802,A -85,B 0,C 180,E1 -17786.012,E2 -17786.012} C_VEL
LIN {X 0,Y 422.375,Z 604.806,A -85,B 0,C 180,E1 -17789.063,E2 -17789.063} C_VEL
LIN {X 0,Y 422.404,Z 604.804,A -85,B 0,C 180,E1 -17792.335,E2 -17792.335} C_VEL
LIN {X 0,Y 422.4,Z 604.802,A -85,B 0,C 180,E1 -17795.789,E2 -17795.789} C_VEL
LIN {X 0,Y 422.426,Z 604.804,A -85,B 0,C 180,E1 -17798.605,E2 -17798.605} C_VEL
LIN {X 0,Y 422.42,Z 604.9,A -85,B 0,C 180,E1 -17799.685,E2 -17799.685} C_VEL
LIN {X 0,Y 424.017,Z 610.994,A -85,B 0,C 180,E1 -17802.205,E2 -17802.205} C_VEL
LIN {X 0,Y 425.892,Z 619.213,A -85,B 0,C 180,E1 -17805.231,E2 -17805.231} C_VEL
LIN {X 0,Y 427.249,Z 626.603,A -85,B 0,C 180,E1 -17807.694,E2 -17807.694} C_VEL
LIN {X 0,Y 427.644,Z 628.846,A -85,B 0,C 180,E1 -17808.395,E2 -17808.395} C_VEL
LIN {X 0,Y 430.864,Z 637.437,A -85,B 0,C 180,E1 -17808.944,E2 -17808.944} C_VEL
LIN {X 0,Y 434.972,Z 654.38,A -85,B 0,C 180,E1 -17809.781,E2 -17809.781} C_VEL
LIN {X 0,Y 435.995,Z 660.127,A -85,B 0,C 180,E1 -17810.03,E2 -17810.03} C_VEL
LIN {X 0,Y 432.464,Z 734.226,A -85,B 0,C 180,E1 -17811.794,E2 -17811.794} C_VEL
LIN {X 0,Y 431.749,Z 744.993,A -85,B 0,C 180,E1 -17812.154,E2 -17812.154} C_VEL
LIN {X 0,Y 431.103,Z 754.518,A -85,B 0,C 180,E1 -17812.59,E2 -17812.59} C_VEL
LIN {X 0,Y 430.363,Z 763.434,A -85,B 0,C 180,E1 -17813.094,E2 -17813.094} C_VEL
LIN {X 0,Y 429.345,Z 773.51,A -85,B 0,C 180,E1 -17813.795,E2 -17813.795} C_VEL
LIN {X 0,Y 428.358,Z 782.958,A -85,B 0,C 180,E1 -17814.605,E2 -17814.605} C_VEL
LIN {X 0,Y 427.222,Z 792.006,A -85,B 0,C 180,E1 -17815.533,E2 -17815.533} C_VEL
LIN {X 0,Y 426.159,Z 799.74,A -85,B 0,C 180,E1 -17816.466,E2 -17816.466} C_VEL
LIN {X 0,Y 424.897,Z 807.843,A -85,B 0,C 180,E1 -17817.638,E2 -17817.638} C_VEL
LIN {X 0,Y 423.741,Z 814.619,A -85,B 0,C 180,E1 -17818.816,E2 -17818.816} C_VEL
LIN {X 0,Y 422.857,Z 820.256,A -85,B 0,C 180,E1 -17820,E2 -17820} C_VEL
LIN {X 0,Y 421.981,Z 825.719,A -85,B 0,C 180,E1 -17821.426,E2 -17821.426} C_VEL
LIN {X 0,Y 421.47,Z 828.785,A -85,B 0,C 180,E1 -17822.381,E2 -17822.381} C_VEL
LIN {X 0,Y 421.047,Z 832.3,A -85,B 0,C 180,E1 -17823.815,E2 -17823.815} C_VEL
LIN {X 0,Y 420.513,Z 835.346,A -85,B 0,C 180,E1 -17825.735,E2 -17825.735} C_VEL
LIN {X 0,Y 420.285,Z 836.316,A -85,B 0,C 180,E1 -17826.699,E2 -17826.699} C_VEL
LIN {X 0,Y 420.084,Z 836.775,A -85,B 0,C 180,E1 -17828.63,E2 -17828.63} C_VEL
LIN {X 0,Y 420.084,Z 836.385,A -85,B 0,C 180,E1 -17829.598,E2 -17829.598} C_VEL
LIN {X 0,Y 420.012,Z 834.232,A -85,B 0,C 180,E1 -17831.544,E2 -17831.544} C_VEL
LIN {X 0,Y 420.089,Z 831.395,A -85,B 0,C 180,E1 -17833.008,E2 -17833.008} C_VEL
LIN {X 0,Y 420.326,Z 827.42,A -85,B 0,C 180,E1 -17834.475,E2 -17834.475} C_VEL
LIN {X 0,Y 420.525,Z 822.153,A -85,B 0,C 180,E1 -17835.952,E2 -17835.952} C_VEL
LIN {X 0,Y 420.8,Z 816.701,A -85,B 0,C 180,E1 -17837.185,E2 -17837.185} C_VEL
LIN {X 0,Y 421.105,Z 810.055,A -85,B 0,C 180,E1 -17838.423,E2 -17838.423} C_VEL
LIN {X 0,Y 421.486,Z 803.811,A -85,B 0,C 180,E1 -17839.412,E2 -17839.412} C_VEL
LIN {X 0,Y 421.993,Z 794.292,A -85,B 0,C 180,E1 -17840.653,E2 -17840.653} C_VEL
LIN {X 0,Y 422.405,Z 786.323,A -85,B 0,C 180,E1 -17841.528,E2 -17841.528} C_VEL
LIN {X 0,Y 422.955,Z 776.946,A -85,B 0,C 180,E1 -17842.389,E2 -17842.389} C_VEL
LIN {X 0,Y 423.468,Z 767.173,A -85,B 0,C 180,E1 -17843.131,E2 -17843.131} C_VEL
LIN {X 0,Y 423.978,Z 755.975,A -85,B 0,C 180,E1 -17843.811,E2 -17843.811} C_VEL
LIN {X 0,Y 424.231,Z 745.348,A -85,B 0,C 180,E1 -17844.314,E2 -17844.314} C_VEL
LIN {X 0,Y 424.591,Z 734.481,A -85,B 0,C 180,E1 -17844.692,E2 -17844.692} C_VEL
LIN {X 0,Y 425.286,Z 708.743,A -85,B 0,C 180,E1 -17845.278,E2 -17845.278} C_VEL
LIN {X 0,Y 426.344,Z 652.491,A -85,B 0,C 180,E1 -17846.51,E2 -17846.51} C_VEL
LIN {X 0,Y 423.076,Z 626.058,A -85,B 0,C 180,E1 -17847.196,E2 -17847.196} C_VEL
LIN {X 0,Y 423.917,Z 614.461,A -85,B 0,C 180,E1 -17849.958,E2 -17849.958} C_VEL
LIN {X 0,Y 423.15,Z 608.544,A -85,B 0,C 180,E1 -17851.427,E2 -17851.427} C_VEL
LIN {X 0,Y 422.47,Z 604.791,A -85,B 0,C 180,E1 -17852.435,E2 -17852.435} C_VEL
LIN {X 0,Y 422.396,Z 604.801,A -85,B 0,C 180,E1 -17855.654,E2 -17855.654} C_VEL
LIN {X 0,Y 422.37,Z 604.801,A -85,B 0,C 180,E1 -17859.063,E2 -17859.063} C_VEL
LIN {X 0,Y 422.361,Z 604.806,A -85,B 0,C 180,E1 -17861.73,E2 -17861.73} C_VEL
LIN {X 0,Y 422.374,Z 604.802,A -85,B 0,C 180,E1 -17864.513,E2 -17864.513} C_VEL
LIN {X 0,Y 422.385,Z 604.799,A -85,B 0,C 180,E1 -17867.163,E2 -17867.163} C_VEL
LIN {X 0,Y 422.383,Z 604.803,A -85,B 0,C 180,E1 -17869.713,E2 -17869.713} C_VEL
LIN {X 0,Y 422.354,Z 604.803,A -85,B 0,C 180,E1 -17872.753,E2 -17872.753} C_VEL
LIN {X 0,Y 422.38,Z 604.803,A -85,B 0,C 180,E1 -17875.679,E2 -17875.679} C_VEL
LIN {X 0,Y 422.37,Z 604.801,A -85,B 0,C 180,E1 -17879.063,E2 -17879.063} C_VEL
LIN {X 0,Y 422.398,Z 604.801,A -85,B 0,C 180,E1 -17882.334,E2 -17882.334} C_VEL
LIN {X 0,Y 422.394,Z 604.803,A -85,B 0,C 180,E1 -17885.789,E2 -17885.789} C_VEL
LIN {X 0,Y 422.42,Z 604.796,A -85,B 0,C 180,E1 -17888.605,E2 -17888.605} C_VEL
LIN {X 0,Y 422.432,Z 604.796,A -85,B 0,C 180,E1 -17891.636,E2 -17891.636} C_VEL
LIN {X 0,Y 422.505,Z 604.785,A -85,B 0,C 180,E1 -17894.618,E2 -17894.618} C_VEL
LIN {X 0,Y 422.562,Z 604.779,A -85,B 0,C 180,E1 -17898.526,E2 -17898.526} C_VEL
LIN {X 0,Y 422.61,Z 604.774,A -85,B 0,C 180,E1 -17902.38,E2 -17902.38} C_VEL
LIN {X 0,Y 422.735,Z 604.756,A -85,B 0,C 180,E1 -17905.248,E2 -17905.248} C_VEL
LIN {X 0,Y 422.545,Z 604.786,A -85,B 0,C 180,E1 -17908.1,E2 -17908.1} C_VEL
LIN {X 0,Y 422.716,Z 604.766,A -85,B 0,C 180,E1 -17910,E2 -17910} C_VEL
LIN {X 0,Y 422.678,Z 604.768,A -85,B 0,C 180,E1 -17913.801,E2 -17913.801} C_VEL
LIN {X 0,Y 422.634,Z 604.769,A -85,B 0,C 180,E1 -17916.662,E2 -17916.662} C_VEL
LIN {X 0,Y 422.521,Z 604.784,A -85,B 0,C 180,E1 -17919.542,E2 -17919.542} C_VEL
LIN {X 0,Y 422.517,Z 604.785,A -85,B 0,C 180,E1 -17922.445,E2 -17922.445} C_VEL
LIN {X 0,Y 422.479,Z 604.794,A -85,B 0,C 180,E1 -17925.931,E2 -17925.931} C_VEL
LIN {X 0,Y 422.437,Z 604.794,A -85,B 0,C 180,E1 -17929.367,E2 -17929.367} C_VEL
LIN {X 0,Y 422.397,Z 604.8,A -85,B 0,C 180,E1 -17932.42,E2 -17932.42} C_VEL
LIN {X 0,Y 422.386,Z 604.801,A -85,B 0,C 180,E1 -17935.541,E2 -17935.541} C_VEL
LIN {X 0,Y 422.393,Z 604.799,A -85,B 0,C 180,E1 -17938.744,E2 -17938.744} C_VEL
LIN {X 0,Y 422.414,Z 604.8,A -85,B 0,C 180,E1 -17942.256,E2 -17942.256} C_VEL
LIN {X 0,Y 422.431,Z 604.797,A -85,B 0,C 180,E1 -17945.662,E2 -17945.662} C_VEL
LIN {X 0,Y 422.416,Z 604.795,A -85,B 0,C 180,E1 -17949.058,E2 -17949.058} C_VEL
LIN {X 0,Y 422.383,Z 604.799,A -85,B 0,C 180,E1 -17952.836,E2 -17952.836} C_VEL
LIN {X 0,Y 422.383,Z 604.805,A -85,B 0,C 180,E1 -17955.854,E2 -17955.854} C_VEL
LIN {X 0,Y 422.361,Z 604.805,A -85,B 0,C 180,E1 -17958.444,E2 -17958.444} C_VEL
LIN {X 0,Y 422.424,Z 604.795,A -85,B 0,C 180,E1 -17961.199,E2 -17961.199} C_VEL
LIN {X 0,Y 422.39,Z 604.803,A -85,B 0,C 180,E1 -17962.282,E2 -17962.282} C_VEL
LIN {X 0,Y 421.706,Z 604.884,A -85,B 0,C 180,E1 -17963.078,E2 -17963.078} C_VEL
LIN {X 0,Y 418.857,Z 605.242,A -85,B 0,C 180,E1 -17964.373,E2 -17964.373} C_VEL
LIN {X 0,Y 416.446,Z 605.545,A -85,B 0,C 180,E1 -17965.417,E2 -17965.417} C_VEL
LIN {X 0,Y 415.398,Z 605.674,A -85,B 0,C 180,E1 -17966.225,E2 -17966.225} C_VEL
LIN {X 0,Y 415.304,Z 605.683,A -85,B 0,C 180,E1 -17966.498,E2 -17966.498} C_VEL
LIN {X 0,Y 415.359,Z 605.677,A -85,B 0,C 180,E1 -17969.609,E2 -17969.609} C_VEL
LIN {X 0,Y 415.336,Z 605.677,A -85,B 0,C 180,E1 -17972.914,E2 -17972.914} C_VEL
LIN {X 0,Y 415.353,Z 605.681,A -85,B 0,C 180,E1 -17976.126,E2 -17976.126} C_VEL
LIN {X 0,Y 415.357,Z 605.675,A -85,B 0,C 180,E1 -17979.26,E2 -17979.26} C_VEL
LIN {X 0,Y 415.391,Z 605.671,A -85,B 0,C 180,E1 -17981.314,E2 -17981.314} C_VEL
LIN {X 0,Y 415.411,Z 605.671,A -85,B 0,C 180,E1 -17984.349,E2 -17984.349} C_VEL
LIN {X 0,Y 415.5,Z 605.663,A -85,B 0,C 180,E1 -17987.892,E2 -17987.892} C_VEL
LIN {X 0,Y 415.544,Z 605.652,A -85,B 0,C 180,E1 -17991.275,E2 -17991.275} C_VEL
LIN {X 0,Y 415.648,Z 605.643,A -85,B 0,C 180,E1 -17994.197,E2 -17994.197} C_VEL
LIN {X 0,Y 415.624,Z 605.641,A -85,B 0,C 180,E1 -17997.102,E2 -17997.102} C_VEL
LIN {X 0,Y 415.671,Z 605.643,A -85,B 0,C 180,E1 -18000,E2 -18000} C_VEL
LIN {X 0,Y 415.639,Z 605.645,A -85,B 0,C 180,E1 -18003.865,E2 -18003.865} C_VEL
LIN {X 0,Y 415.601,Z 605.645,A -85,B 0,C 180,E1 -18006.776,E2 -18006.776} C_VEL
LIN {X 0,Y 415.484,Z 605.663,A -85,B 0,C 180,E1 -18009.706,E2 -18009.706} C_VEL
LIN {X 0,Y 415.459,Z 605.663,A -85,B 0,C 180,E1 -18012.661,E2 -18012.661} C_VEL
LIN {X 0,Y 415.375,Z 605.68,A -85,B 0,C 180,E1 -18016.016,E2 -18016.016} C_VEL
LIN {X 0,Y 415.375,Z 605.673,A -85,B 0,C 180,E1 -18019.209,E2 -18019.209} C_VEL
LIN {X 0,Y 415.346,Z 605.683,A -85,B 0,C 180,E1 -18021.948,E2 -18021.948} C_VEL
LIN {X 0,Y 415.34,Z 605.677,A -85,B 0,C 180,E1 -18024.936,E2 -18024.936} C_VEL
LIN {X 0,Y 415.348,Z 605.681,A -85,B 0,C 180,E1 -18028.177,E2 -18028.177} C_VEL
LIN {X 0,Y 415.295,Z 605.684,A -85,B 0,C 180,E1 -18031.524,E2 -18031.524} C_VEL
LIN {X 0,Y 415.31,Z 605.68,A -85,B 0,C 180,E1 -18034.99,E2 -18034.99} C_VEL
LIN {X 0,Y 415.312,Z 605.683,A -85,B 0,C 180,E1 -18037.564,E2 -18037.564} C_VEL
LIN {X 0,Y 415.271,Z 605.685,A -85,B 0,C 180,E1 -18041.134,E2 -18041.134} C_VEL
LIN {X 0,Y 415.304,Z 605.686,A -85,B 0,C 180,E1 -18043.749,E2 -18043.749} C_VEL
LIN {X 0,Y 415.299,Z 605.684,A -85,B 0,C 180,E1 -18046.489,E2 -18046.489} C_VEL
LIN {X 0,Y 415.274,Z 605.691,A -85,B 0,C 180,E1 -18050.138,E2 -18050.138} C_VEL
LIN {X 0,Y 415.302,Z 605.683,A -85,B 0,C 180,E1 -18052.615,E2 -18052.615} C_VEL
LIN {X 0,Y 415.269,Z 605.691,A -85,B 0,C 180,E1 -18056.178,E2 -18056.178} C_VEL
LIN {X 0,Y 415.344,Z 605.679,A -85,B 0,C 180,E1 -18059.607,E2 -18059.607} C_VEL
LIN {X 0,Y 415.324,Z 605.679,A -85,B 0,C 180,E1 -18062.912,E2 -18062.912} C_VEL
LIN {X 0,Y 415.438,Z 605.858,A -85,B 0,C 180,E1 -18063.95,E2 -18063.95} C_VEL
LIN {X 0,Y 417.889,Z 619.815,A -85,B 0,C 180,E1 -18067.203,E2 -18067.203} C_VEL
LIN {X 0,Y 416.938,Z 630.829,A -85,B 0,C 180,E1 -18069.624,E2 -18069.624} C_VEL
LIN {X 0,Y 415.722,Z 644.703,A -85,B 0,C 180,E1 -18072.641,E2 -18072.641} C_VEL
LIN {X 0,Y 418.79,Z 675.658,A -85,B 0,C 180,E1 -18073.43,E2 -18073.43} C_VEL
LIN {X 0,Y 419.122,Z 682.217,A -85,B 0,C 180,E1 -18073.588,E2 -18073.588} C_VEL
LIN {X 0,Y 417.649,Z 750.996,A -85,B 0,C 180,E1 -18075.151,E2 -18075.151} C_VEL
LIN {X 0,Y 417.282,Z 761.132,A -85,B 0,C 180,E1 -18075.479,E2 -18075.479} C_VEL
LIN {X 0,Y 416.91,Z 771.974,A -85,B 0,C 180,E1 -18075.962,E2 -18075.962} C_VEL
LIN {X 0,Y 416.506,Z 781.522,A -85,B 0,C 180,E1 -18076.507,E2 -18076.507} C_VEL
LIN {X 0,Y 415.987,Z 791.752,A -85,B 0,C 180,E1 -18077.232,E2 -18077.232} C_VEL
LIN {X 0,Y 415.487,Z 799.68,A -85,B 0,C 180,E1 -18077.901,E2 -18077.901} C_VEL
LIN {X 0,Y 414.979,Z 809.719,A -85,B 0,C 180,E1 -18078.931,E2 -18078.931} C_VEL
LIN {X 0,Y 414.487,Z 816.784,A -85,B 0,C 180,E1 -18079.779,E2 -18079.779} C_VEL
LIN {X 0,Y 414.013,Z 825.203,A -85,B 0,C 180,E1 -18080.997,E2 -18080.997} C_VEL
LIN {X 0,Y 413.626,Z 832.207,A -85,B 0,C 180,E1 -18082.214,E2 -18082.214} C_VEL
LIN {X 0,Y 413.433,Z 838.055,A -85,B 0,C 180,E1 -18083.434,E2 -18083.434} C_VEL
LIN {X 0,Y 413.283,Z 842.902,A -85,B 0,C 180,E1 -18084.652,E2 -18084.652} C_VEL
LIN {X 0,Y 413.165,Z 847.474,A -85,B 0,C 180,E1 -18086.112,E2 -18086.112} C_VEL
LIN {X 0,Y 413.145,Z 849.863,A -85,B 0,C 180,E1 -18087.085,E2 -18087.085} C_VEL
LIN {X 0,Y 413.127,Z 853.272,A -85,B 0,C 180,E1 -18089.029,E2 -18089.029} C_VEL
LIN {X 0,Y 413.111,Z 854.247,A -85,B 0,C 180,E1 -18090,E2 -18090} C_VEL
LIN {X 0,Y 413.087,Z 855.027,A -85,B 0,C 180,E1 -18091.944,E2 -18091.944} C_VEL
LIN {X 0,Y 413.104,Z 853.939,A -85,B 0,C 180,E1 -18093.889,E2 -18093.889} C_VEL
LIN {X 0,Y 413.235,Z 852.874,A -85,B 0,C 180,E1 -18094.862,E2 -18094.862} C_VEL
LIN {X 0,Y 413.656,Z 849.218,A -85,B 0,C 180,E1 -18096.808,E2 -18096.808} C_VEL
LIN {X 0,Y 414.165,Z 845.297,A -85,B 0,C 180,E1 -18098.265,E2 -18098.265} C_VEL
LIN {X 0,Y 414.828,Z 840.216,A -85,B 0,C 180,E1 -18099.721,E2 -18099.721} C_VEL
LIN {X 0,Y 415.749,Z 835.02,A -85,B 0,C 180,E1 -18100.926,E2 -18100.926} C_VEL
LIN {X 0,Y 416.745,Z 828.783,A -85,B 0,C 180,E1 -18102.128,E2 -18102.128} C_VEL
LIN {X 0,Y 417.838,Z 821.357,A -85,B 0,C 180,E1 -18103.321,E2 -18103.321} C_VEL
LIN {X 0,Y 419.276,Z 812.354,A -85,B 0,C 180,E1 -18104.513,E2 -18104.513} C_VEL
LIN {X 0,Y 420.437,Z 803.852,A -85,B 0,C 180,E1 -18105.46,E2 -18105.46} C_VEL
LIN {X 0,Y 421.767,Z 793.608,A -85,B 0,C 180,E1 -18106.399,E2 -18106.399} C_VEL
LIN {X 0,Y 422.87,Z 784.374,A -85,B 0,C 180,E1 -18107.099,E2 -18107.099} C_VEL
LIN {X 0,Y 423.996,Z 774.005,A -85,B 0,C 180,E1 -18107.734,E2 -18107.734} C_VEL
LIN {X 0,Y 425.084,Z 763.223,A -85,B 0,C 180,E1 -18108.245,E2 -18108.245} C_VEL
LIN {X 0,Y 425.852,Z 752.146,A -85,B 0,C 180,E1 -18108.646,E2 -18108.646} C_VEL
LIN {X 0,Y 427.662,Z 713.68,A -85,B 0,C 180,E1 -18109.594,E2 -18109.594} C_VEL
LIN {X 0,Y 428.994,Z 683.375,A -85,B 0,C 180,E1 -18110.349,E2 -18110.349} C_VEL
LIN {X 0,Y 427.025,Z 669.444,A -85,B 0,C 180,E1 -18110.925,E2 -18110.925} C_VEL
LIN {X 0,Y 423.507,Z 653.118,A -85,B 0,C 180,E1 -18111.72,E2 -18111.72} C_VEL
LIN {X 0,Y 420.805,Z 642.381,A -85,B 0,C 180,E1 -18112.336,E2 -18112.336} C_VEL
LIN {X 0,Y 421.806,Z 635.648,A -85,B 0,C 180,E1 -18114.032,E2 -18114.032} C_VEL
LIN {X 0,Y 420.681,Z 628.074,A -85,B 0,C 180,E1 -18116.253,E2 -18116.253} C_VEL
LIN {X 0,Y 419.353,Z 621.252,A -85,B 0,C 180,E1 -18118.427,E2 -18118.427} C_VEL
LIN {X 0,Y 417.441,Z 613.598,A -85,B 0,C 180,E1 -18121.157,E2 -18121.157} C_VEL
LIN {X 0,Y 415.338,Z 605.681,A -85,B 0,C 180,E1 -18124.388,E2 -18124.388} C_VEL
LIN {X 0,Y 415.321,Z 605.677,A -85,B 0,C 180,E1 -18127.565,E2 -18127.565} C_VEL
LIN {X 0,Y 415.289,Z 605.681,A -85,B 0,C 180,E1 -18131.132,E2 -18131.132} C_VEL
LIN {X 0,Y 415.314,Z 605.679,A -85,B 0,C 180,E1 -18133.748,E2 -18133.748} C_VEL
LIN {X 0,Y 415.36,Z 605.68,A -85,B 0,C 180,E1 -18136.48,E2 -18136.48} C_VEL
LIN {X 0,Y 415.344,Z 605.681,A -85,B 0,C 180,E1 -18140.145,E2 -18140.145} C_VEL
LIN {X 0,Y 415.331,Z 605.683,A -85,B 0,C 180,E1 -18143.824,E2 -18143.824} C_VEL
LIN {X 0,Y 415.332,Z 605.68,A -85,B 0,C 180,E1 -18146.183,E2 -18146.183} C_VEL
LIN {X 0,Y 415.364,Z 605.676,A -85,B 0,C 180,E1 -18149.609,E2 -18149.609} C_VEL
LIN {X 0,Y 415.342,Z 605.68,A -85,B 0,C 180,E1 -18152.913,E2 -18152.913} C_VEL
LIN {X 0,Y 415.358,Z 605.68,A -85,B 0,C 180,E1 -18156.126,E2 -18156.126} C_VEL
LIN {X 0,Y 415.375,Z 605.722,A -85,B 0,C 180,E1 -18158.743,E2 -18158.743} C_VEL
LIN {X 0,Y 417.292,Z 612.983,A -85,B 0,C 180,E1 -18161.909,E2 -18161.909} C_VEL
LIN {X 0,Y 419.122,Z 621.092,A -85,B 0,C 180,E1 -18164.987,E2 -18164.987} C_VEL
LIN {X 0,Y 420.558,Z 629.061,A -85,B 0,C 180,E1 -18167.715,E2 -18167.715} C_VEL
LIN {X 0,Y 424.524,Z 638.152,A -85,B 0,C 180,E1 -18168.391,E2 -18168.391} C_VEL
LIN {X 0,Y 427.558,Z 649.714,A -85,B 0,C 180,E1 -18169.014,E2 -18169.014} C_VEL
LIN {X 0,Y 429.931,Z 661.13,A -85,B 0,C 180,E1 -18169.551,E2 -18169.551} C_VEL
LIN {X 0,Y 426.169,Z 735.126,A -85,B 0,C 180,E1 -18171.374,E2 -18171.374} C_VEL
LIN {X 0,Y 425.402,Z 745.901,A -85,B 0,C 180,E1 -18171.748,E2 -18171.748} C_VEL
LIN {X 0,Y 424.65,Z 756.228,A -85,B 0,C 180,E1 -18172.241,E2 -18172.241} C_VEL
LIN {X 0,Y 423.788,Z 765.534,A -85,B 0,C 180,E1 -18172.796,E2 -18172.796} C_VEL
LIN {X 0,Y 422.809,Z 774.688,A -85,B 0,C 180,E1 -18173.46,E2 -18173.46} C_VEL
LIN {X 0,Y 421.785,Z 783.978,A -85,B 0,C 180,E1 -18174.281,E2 -18174.281} C_VEL
LIN {X 0,Y 420.582,Z 792.908,A -85,B 0,C 180,E1 -18175.223,E2 -18175.223} C_VEL
LIN {X 0,Y 419.443,Z 800.494,A -85,B 0,C 180,E1 -18176.17,E2 -18176.17} C_VEL
LIN {X 0,Y 418.382,Z 807.041,A -85,B 0,C 180,E1 -18177.121,E2 -18177.121} C_VEL
LIN {X 0,Y 417.17,Z 813.951,A -85,B 0,C 180,E1 -18178.316,E2 -18178.316} C_VEL
LIN {X 0,Y 416.135,Z 819.768,A -85,B 0,C 180,E1 -18179.517,E2 -18179.517} C_VEL
LIN {X 0,Y 415.219,Z 825.369,A -85,B 0,C 180,E1 -18180.966,E2 -18180.966} C_VEL
LIN {X 0,Y 414.383,Z 829.784,A -85,B 0,C 180,E1 -18182.422,E2 -18182.422} C_VEL
LIN {X 0,Y 413.949,Z 833.077,A -85,B 0,C 180,E1 -18183.881,E2 -18183.881} C_VEL
LIN {X 0,Y 413.484,Z 835.365,A -85,B 0,C 180,E1 -18185.417,E2 -18185.417} C_VEL
LIN {X 0,Y 413.169,Z 836.68,A -85,B 0,C 180,E1 -18186.815,E2 -18186.815} C_VEL
LIN {X 0,Y 413.008,Z 836.97,A -85,B 0,C 180,E1 -18187.797,E2 -18187.797} C_VEL
LIN {X 0,Y 412.997,Z 836.374,A -85,B 0,C 180,E1 -18189.764,E2 -18189.764} C_VEL
LIN {X 0,Y 412.963,Z 835.306,A -85,B 0,C 180,E1 -18190.753,E2 -18190.753} C_VEL
LIN {X 0,Y 412.957,Z 832.003,A -85,B 0,C 180,E1 -18192.738,E2 -18192.738} C_VEL
LIN {X 0,Y 413.189,Z 828.167,A -85,B 0,C 180,E1 -18194.229,E2 -18194.229} C_VEL
LIN {X 0,Y 413.383,Z 823.043,A -85,B 0,C 180,E1 -18195.73,E2 -18195.73} C_VEL
LIN {X 0,Y 413.71,Z 816.484,A -85,B 0,C 180,E1 -18197.234,E2 -18197.234} C_VEL
LIN {X 0,Y 414.013,Z 810.272,A -85,B 0,C 180,E1 -18198.407,E2 -18198.407} C_VEL
LIN {X 0,Y 414.423,Z 803.406,A -85,B 0,C 180,E1 -18199.5,E2 -18199.5} C_VEL
LIN {X 0,Y 414.899,Z 794.856,A -85,B 0,C 180,E1 -18200.635,E2 -18200.635} C_VEL
LIN {X 0,Y 415.367,Z 785.705,A -85,B 0,C 180,E1 -18201.646,E2 -18201.646} C_VEL
LIN {X 0,Y 415.86,Z 777.071,A -85,B 0,C 180,E1 -18202.449,E2 -18202.449} C_VEL
LIN {X 0,Y 416.362,Z 768.008,A -85,B 0,C 180,E1 -18203.156,E2 -18203.156} C_VEL
LIN {X 0,Y 416.856,Z 756.971,A -85,B 0,C 180,E1 -18203.848,E2 -18203.848} C_VEL
LIN {X 0,Y 417.154,Z 745.881,A -85,B 0,C 180,E1 -18204.39,E2 -18204.39} C_VEL
LIN {X 0,Y 417.555,Z 734.55,A -85,B 0,C 180,E1 -18204.795,E2 -18204.795} C_VEL
LIN {X 0,Y 418.239,Z 709.227,A -85,B 0,C 180,E1 -18205.39,E2 -18205.39} C_VEL
LIN {X 0,Y 419.324,Z 652.863,A -85,B 0,C 180,E1 -18206.662,E2 -18206.662} C_VEL
LIN {X 0,Y 416.191,Z 627.523,A -85,B 0,C 180,E1 -18207.323,E2 -18207.323} C_VEL
LIN {X 0,Y 416.084,Z 626.113,A -85,B 0,C 180,E1 -18207.389,E2 -18207.389} C_VEL
LIN {X 0,Y 416.871,Z 615.366,A -85,B 0,C 180,E1 -18209.991,E2 -18209.991} C_VEL
LIN {X 0,Y 416.141,Z 609.562,A -85,B 0,C 180,E1 -18211.452,E2 -18211.452} C_VEL
LIN {X 0,Y 415.427,Z 605.668,A -85,B 0,C 180,E1 -18212.5,E2 -18212.5} C_VEL
LIN {X 0,Y 415.328,Z 605.684,A -85,B 0,C 180,E1 -18216.176,E2 -18216.176} C_VEL
LIN {X 0,Y 415.33,Z 605.684,A -85,B 0,C 180,E1 -18219.855,E2 -18219.855} C_VEL
LIN {X 0,Y 415.357,Z 605.677,A -85,B 0,C 180,E1 -18223.519,E2 -18223.519} C_VEL
LIN {X 0,Y 415.357,Z 605.677,A -85,B 0,C 180,E1 -18226.48,E2 -18226.48} C_VEL
LIN {X 0,Y 415.329,Z 605.684,A -85,B 0,C 180,E1 -18230.144,E2 -18230.144} C_VEL
LIN {X 0,Y 415.33,Z 605.683,A -85,B 0,C 180,E1 -18233.824,E2 -18233.824} C_VEL
LIN {X 0,Y 415.327,Z 605.684,A -85,B 0,C 180,E1 -18236.183,E2 -18236.183} C_VEL
LIN {X 0,Y 415.358,Z 605.677,A -85,B 0,C 180,E1 -18239.608,E2 -18239.608} C_VEL
LIN {X 0,Y 415.335,Z 605.677,A -85,B 0,C 180,E1 -18242.913,E2 -18242.913} C_VEL
LIN {X 0,Y 415.352,Z 605.681,A -85,B 0,C 180,E1 -18246.125,E2 -18246.125} C_VEL
LIN {X 0,Y 415.355,Z 605.675,A -85,B 0,C 180,E1 -18249.259,E2 -18249.259} C_VEL
LIN {X 0,Y 415.377,Z 605.676,A -85,B 0,C 180,E1 -18252.33,E2 -18252.33} C_VEL
LIN {X 0,Y 415.436,Z 605.666,A -85,B 0,C 180,E1 -18255.35,E2 -18255.35} C_VEL
LIN {X 0,Y 415.512,Z 605.659,A -85,B 0,C 180,E1 -18258.329,E2 -18258.329} C_VEL
LIN {X 0,Y 415.565,Z 605.653,A -85,B 0,C 180,E1 -18262.25,E2 -18262.25} C_VEL
LIN {X 0,Y 415.688,Z 605.634,A -85,B 0,C 180,E1 -18265.167,E2 -18265.167} C_VEL
LIN {X 0,Y 415.517,Z 605.661,A -85,B 0,C 180,E1 -18268.068,E2 -18268.068} C_VEL
LIN {X 0,Y 415.669,Z 605.643,A -85,B 0,C 180,E1 -18270,E2 -18270} C_VEL
LIN {X 0,Y 415.644,Z 605.645,A -85,B 0,C 180,E1 -18273.865,E2 -18273.865} C_VEL
LIN {X 0,Y 415.596,Z 605.645,A -85,B 0,C 180,E1 -18276.775,E2 -18276.775} C_VEL
LIN {X 0,Y 415.48,Z 605.663,A -85,B 0,C 180,E1 -18279.705,E2 -18279.705} C_VEL
LIN {X 0,Y 415.461,Z 605.662,A -85,B 0,C 180,E1 -18282.66,E2 -18282.66} C_VEL
LIN {X 0,Y 415.443,Z 605.671,A -85,B 0,C 180,E1 -18286.051,E2 -18286.051} C_VEL
LIN {X 0,Y 415.377,Z 605.676,A -85,B 0,C 180,E1 -18289.71,E2 -18289.71} C_VEL
LIN {X 0,Y 415.331,Z 605.678,A -85,B 0,C 180,E1 -18292.823,E2 -18292.823} C_VEL
LIN {X 0,Y 415.341,Z 605.684,A -85,B 0,C 180,E1 -18296.006,E2 -18296.006} C_VEL
LIN {X 0,Y 415.344,Z 605.677,A -85,B 0,C 180,E1 -18299.279,E2 -18299.279} C_VEL
LIN {X 0,Y 415.353,Z 605.676,A -85,B 0,C 180,E1 -18302.659,E2 -18302.659} C_VEL
LIN {X 0,Y 415.401,Z 605.675,A -85,B 0,C 180,E1 -18306.169,E2 -18306.169} C_VEL
LIN {X 0,Y 415.379,Z 605.672,A -85,B 0,C 180,E1 -18309.133,E2 -18309.133} C_VEL
LIN {X 0,Y 415.317,Z 605.682,A -85,B 0,C 180,E1 -18312.424,E2 -18312.424} C_VEL
LIN {X 0,Y 415.341,Z 605.677,A -85,B 0,C 180,E1 -18315.097,E2 -18315.097} C_VEL
LIN {X 0,Y 415.312,Z 605.687,A -85,B 0,C 180,E1 -18317.909,E2 -18317.909} C_VEL
LIN {X 0,Y 415.376,Z 605.673,A -85,B 0,C 180,E1 -18321.397,E2 -18321.397} C_VEL
LIN {X 0,Y 415.35,Z 605.675,A -85,B 0,C 180,E1 -18325.015,E2 -18325.015} C_VEL
LIN {X 0,Y 415.304,Z 605.683,A -85,B 0,C 180,E1 -18326.498,E2 -18326.498} C_VEL
LIN {X 0,Y 414.613,Z 605.769,A -85,B 0,C 180,E1 -18327.308,E2 -18327.308} C_VEL
LIN {X 0,Y 411.75,Z 606.125,A -85,B 0,C 180,E1 -18328.624,E2 -18328.624} C_VEL
LIN {X 0,Y 409.362,Z 606.425,A -85,B 0,C 180,E1 -18329.687,E2 -18329.687} C_VEL
LIN {X 0,Y 408.365,Z 606.548,A -85,B 0,C 180,E1 -18330.508,E2 -18330.508} C_VEL
LIN {X 0,Y 408.298,Z 606.554,A -85,B 0,C 180,E1 -18330.786,E2 -18330.786} C_VEL
LIN {X 0,Y 408.338,Z 606.551,A -85,B 0,C 180,E1 -18333.514,E2 -18333.514} C_VEL
LIN {X 0,Y 408.301,Z 606.554,A -85,B 0,C 180,E1 -18336.761,E2 -18336.761} C_VEL
LIN {X 0,Y 408.378,Z 606.545,A -85,B 0,C 180,E1 -18340.622,E2 -18340.622} C_VEL
LIN {X 0,Y 408.362,Z 606.553,A -85,B 0,C 180,E1 -18344.072,E2 -18344.072} C_VEL
LIN {X 0,Y 408.466,Z 606.538,A -85,B 0,C 180,E1 -18347.808,E2 -18347.808} C_VEL
LIN {X 0,Y 408.482,Z 606.531,A -85,B 0,C 180,E1 -18351.123,E2 -18351.123} C_VEL
LIN {X 0,Y 408.615,Z 606.521,A -85,B 0,C 180,E1 -18354.097,E2 -18354.097} C_VEL
LIN {X 0,Y 408.605,Z 606.516,A -85,B 0,C 180,E1 -18357.052,E2 -18357.052} C_VEL
LIN {X 0,Y 408.624,Z 606.521,A -85,B 0,C 180,E1 -18360,E2 -18360} C_VEL
LIN {X 0,Y 408.606,Z 606.522,A -85,B 0,C 180,E1 -18363.932,E2 -18363.932} C_VEL
LIN {X 0,Y 408.553,Z 606.522,A -85,B 0,C 180,E1 -18366.893,E2 -18366.893} C_VEL
LIN {X 0,Y 408.428,Z 606.544,A -85,B 0,C 180,E1 -18369.875,E2 -18369.875} C_VEL
LIN {X 0,Y 408.423,Z 606.538,A -85,B 0,C 180,E1 -18372.883,E2 -18372.883} C_VEL
LIN {X 0,Y 408.324,Z 606.557,A -85,B 0,C 180,E1 -18376.131,E2 -18376.131} C_VEL
LIN {X 0,Y 408.319,Z 606.552,A -85,B 0,C 180,E1 -18379.354,E2 -18379.354} C_VEL
LIN {X 0,Y 408.297,Z 606.559,A -85,B 0,C 180,E1 -18382.174,E2 -18382.174} C_VEL
LIN {X 0,Y 408.305,Z 606.554,A -85,B 0,C 180,E1 -18385.396,E2 -18385.396} C_VEL
LIN {X 0,Y 408.312,Z 606.552,A -85,B 0,C 180,E1 -18388.969,E2 -18388.969} C_VEL
LIN {X 0,Y 408.23,Z 606.568,A -85,B 0,C 180,E1 -18392.134,E2 -18392.134} C_VEL
LIN {X 0,Y 408.287,Z 606.559,A -85,B 0,C 180,E1 -18395.683,E2 -18395.683} C_VEL
LIN {X 0,Y 408.254,Z 606.565,A -85,B 0,C 180,E1 -18398.145,E2 -18398.145} C_VEL
LIN {X 0,Y 408.235,Z 606.569,A -85,B 0,C 180,E1 -18402.002,E2 -18402.002} C_VEL
LIN {X 0,Y 408.27,Z 606.558,A -85,B 0,C 180,E1 -18405.299,E2 -18405.299} C_VEL
LIN {X 0,Y 408.233,Z 606.562,A -85,B 0,C 180,E1 -18409.021,E2 -18409.021} C_VEL
LIN {X 0,Y 408.255,Z 606.565,A -85,B 0,C 180,E1 -18412.113,E2 -18412.113} C_VEL
LIN {X 0,Y 408.255,Z 606.561,A -85,B 0,C 180,E1 -18415.516,E2 -18415.516} C_VEL
LIN {X 0,Y 408.262,Z 606.558,A -85,B 0,C 180,E1 -18419.075,E2 -18419.075} C_VEL
LIN {X 0,Y 408.281,Z 606.559,A -85,B 0,C 180,E1 -18422.406,E2 -18422.406} C_VEL
LIN {X 0,Y 408.407,Z 606.748,A -85,B 0,C 180,E1 -18423.861,E2 -18423.861} C_VEL
LIN {X 0,Y 410.756,Z 620.216,A -85,B 0,C 180,E1 -18427.049,E2 -18427.049} C_VEL
LIN {X 0,Y 410.493,Z 625.388,A -85,B 0,C 180,E1 -18428.215,E2 -18428.215} C_VEL
LIN {X 0,Y 408.848,Z 642.586,A -85,B 0,C 180,E1 -18432.039,E2 -18432.039} C_VEL
LIN {X 0,Y 408.697,Z 644.554,A -85,B 0,C 180,E1 -18432.475,E2 -18432.475} C_VEL
LIN {X 0,Y 411.676,Z 675.827,A -85,B 0,C 180,E1 -18433.289,E2 -18433.289} C_VEL
LIN {X 0,Y 412.114,Z 681.377,A -85,B 0,C 180,E1 -18433.43,E2 -18433.43} C_VEL
LIN {X 0,Y 410.604,Z 750.804,A -85,B 0,C 180,E1 -18435.048,E2 -18435.048} C_VEL
LIN {X 0,Y 410.219,Z 760.912,A -85,B 0,C 180,E1 -18435.381,E2 -18435.381} C_VEL
LIN {X 0,Y 409.889,Z 771.187,A -85,B 0,C 180,E1 -18435.843,E2 -18435.843} C_VEL
LIN {X 0,Y 409.457,Z 780.848,A -85,B 0,C 180,E1 -18436.396,E2 -18436.396} C_VEL
LIN {X 0,Y 408.944,Z 791.173,A -85,B 0,C 180,E1 -18437.135,E2 -18437.135} C_VEL
LIN {X 0,Y 408.301,Z 800.7,A -85,B 0,C 180,E1 -18437.966,E2 -18437.966} C_VEL
LIN {X 0,Y 407.917,Z 809.271,A -85,B 0,C 180,E1 -18438.862,E2 -18438.862} C_VEL
LIN {X 0,Y 407.371,Z 817.258,A -85,B 0,C 180,E1 -18439.849,E2 -18439.849} C_VEL
LIN {X 0,Y 406.887,Z 825.576,A -85,B 0,C 180,E1 -18441.087,E2 -18441.087} C_VEL
LIN {X 0,Y 406.535,Z 832.497,A -85,B 0,C 180,E1 -18442.327,E2 -18442.327} C_VEL
LIN {X 0,Y 406.322,Z 838.263,A -85,B 0,C 180,E1 -18443.567,E2 -18443.567} C_VEL
LIN {X 0,Y 406.199,Z 842.213,A -85,B 0,C 180,E1 -18444.558,E2 -18444.558} C_VEL
LIN {X 0,Y 406.091,Z 846.93,A -85,B 0,C 180,E1 -18446.044,E2 -18446.044} C_VEL
LIN {X 0,Y 406.064,Z 849.335,A -85,B 0,C 180,E1 -18447.034,E2 -18447.034} C_VEL
LIN {X 0,Y 406.059,Z 852.94,A -85,B 0,C 180,E1 -18449.012,E2 -18449.012} C_VEL
LIN {X 0,Y 405.999,Z 854.567,A -85,B 0,C 180,E1 -18450.989,E2 -18450.989} C_VEL
LIN {X 0,Y 405.986,Z 854.848,A -85,B 0,C 180,E1 -18451.978,E2 -18451.978} C_VEL
LIN {X 0,Y 406.022,Z 853.929,A -85,B 0,C 180,E1 -18453.957,E2 -18453.957} C_VEL
LIN {X 0,Y 406.149,Z 852.867,A -85,B 0,C 180,E1 -18454.947,E2 -18454.947} C_VEL
LIN {X 0,Y 406.593,Z 849.418,A -85,B 0,C 180,E1 -18456.926,E2 -18456.926} C_VEL
LIN {X 0,Y 407.139,Z 845.604,A -85,B 0,C 180,E1 -18458.409,E2 -18458.409} C_VEL
LIN {X 0,Y 408.015,Z 839.632,A -85,B 0,C 180,E1 -18460.135,E2 -18460.135} C_VEL
LIN {X 0,Y 409.02,Z 834.376,A -85,B 0,C 180,E1 -18461.358,E2 -18461.358} C_VEL
LIN {X 0,Y 410.11,Z 828.096,A -85,B 0,C 180,E1 -18462.578,E2 -18462.578} C_VEL
LIN {X 0,Y 411.244,Z 820.589,A -85,B 0,C 180,E1 -18463.795,E2 -18463.795} C_VEL
LIN {X 0,Y 412.631,Z 812.523,A -85,B 0,C 180,E1 -18464.877,E2 -18464.877} C_VEL
LIN {X 0,Y 414.036,Z 802.858,A -85,B 0,C 180,E1 -18465.957,E2 -18465.957} C_VEL
LIN {X 0,Y 415.257,Z 793.893,A -85,B 0,C 180,E1 -18466.79,E2 -18466.79} C_VEL
LIN {X 0,Y 416.427,Z 784.747,A -85,B 0,C 180,E1 -18467.498,E2 -18467.498} C_VEL
LIN {X 0,Y 417.72,Z 773.429,A -85,B 0,C 180,E1 -18468.199,E2 -18468.199} C_VEL
LIN {X 0,Y 418.826,Z 762.721,A -85,B 0,C 180,E1 -18468.717,E2 -18468.717} C_VEL
LIN {X 0,Y 419.65,Z 751.739,A -85,B 0,C 180,E1 -18469.121,E2 -18469.121} C_VEL
LIN {X 0,Y 421.627,Z 713.034,A -85,B 0,C 180,E1 -18470.101,E2 -18470.101} C_VEL
LIN {X 0,Y 422.948,Z 684.756,A -85,B 0,C 180,E1 -18470.819,E2 -18470.819} C_VEL
LIN {X 0,Y 421.115,Z 671.558,A -85,B 0,C 180,E1 -18471.376,E2 -18471.376} C_VEL
LIN {X 0,Y 417.65,Z 654.887,A -85,B 0,C 180,E1 -18472.223,E2 -18472.223} C_VEL
LIN {X 0,Y 414.372,Z 642.203,A -85,B 0,C 180,E1 -18472.978,E2 -18472.978} C_VEL
LIN {X 0,Y 415.018,Z 638.596,A -85,B 0,C 180,E1 -18473.895,E2 -18473.895} C_VEL
LIN {X 0,Y 414.435,Z 633.012,A -85,B 0,C 180,E1 -18475.53,E2 -18475.53} C_VEL
LIN {X 0,Y 412.834,Z 624.167,A -85,B 0,C 180,E1 -18478.364,E2 -18478.364} C_VEL
LIN {X 0,Y 411.264,Z 617.605,A -85,B 0,C 180,E1 -18480.727,E2 -18480.727} C_VEL
LIN {X 0,Y 409.244,Z 610.079,A -85,B 0,C 180,E1 -18483.798,E2 -18483.798} C_VEL
LIN {X 0,Y 408.291,Z 606.557,A -85,B 0,C 180,E1 -18485.456,E2 -18485.456} C_VEL
LIN {X 0,Y 408.267,Z 606.552,A -85,B 0,C 180,E1 -18488.144,E2 -18488.144} C_VEL
LIN {X 0,Y 408.252,Z 606.558,A -85,B 0,C 180,E1 -18490.982,E2 -18490.982} C_VEL
LIN {X 0,Y 408.282,Z 606.559,A -85,B 0,C 180,E1 -18494.7,E2 -18494.7} C_VEL
LIN {X 0,Y 408.277,Z 606.56,A -85,B 0,C 180,E1 -18497.537,E2 -18497.537} C_VEL
LIN {X 0,Y 408.302,Z 606.556,A -85,B 0,C 180,E1 -18500.599,E2 -18500.599} C_VEL
LIN {X 0,Y 408.304,Z 606.555,A -85,B 0,C 180,E1 -18504.319,E2 -18504.319} C_VEL
LIN {X 0,Y 408.26,Z 606.561,A -85,B 0,C 180,E1 -18507.869,E2 -18507.869} C_VEL
LIN {X 0,Y 408.323,Z 606.554,A -85,B 0,C 180,E1 -18511.294,E2 -18511.294} C_VEL
LIN {X 0,Y 408.31,Z 606.557,A -85,B 0,C 180,E1 -18514.604,E2 -18514.604} C_VEL
LIN {X 0,Y 408.343,Z 606.692,A -85,B 0,C 180,E1 -18517.762,E2 -18517.762} C_VEL
LIN {X 0,Y 410.248,Z 613.76,A -85,B 0,C 180,E1 -18521.071,E2 -18521.071} C_VEL
LIN {X 0,Y 412.087,Z 621.584,A -85,B 0,C 180,E1 -18524.219,E2 -18524.219} C_VEL
LIN {X 0,Y 413.565,Z 629.448,A -85,B 0,C 180,E1 -18527.016,E2 -18527.016} C_VEL
LIN {X 0,Y 418.569,Z 640.137,A -85,B 0,C 180,E1 -18527.877,E2 -18527.877} C_VEL
LIN {X 0,Y 421.12,Z 649.159,A -85,B 0,C 180,E1 -18528.41,E2 -18528.41} C_VEL
LIN {X 0,Y 423.904,Z 662.298,A -85,B 0,C 180,E1 -18529.064,E2 -18529.064} C_VEL
LIN {X 0,Y 420.004,Z 734.83,A -85,B 0,C 180,E1 -18530.884,E2 -18530.884} C_VEL
LIN {X 0,Y 419.2,Z 745.559,A -85,B 0,C 180,E1 -18531.26,E2 -18531.26} C_VEL
LIN {X 0,Y 418.433,Z 755.606,A -85,B 0,C 180,E1 -18531.744,E2 -18531.744} C_VEL
LIN {X 0,Y 417.55,Z 764.707,A -85,B 0,C 180,E1 -18532.287,E2 -18532.287} C_VEL
LIN {X 0,Y 416.401,Z 775.06,A -85,B 0,C 180,E1 -18533.048,E2 -18533.048} C_VEL
LIN {X 0,Y 415.355,Z 783.825,A -85,B 0,C 180,E1 -18533.828,E2 -18533.828} C_VEL
LIN {X 0,Y 414.252,Z 791.814,A -85,B 0,C 180,E1 -18534.664,E2 -18534.664} C_VEL
LIN {X 0,Y 413.077,Z 799.604,A -85,B 0,C 180,E1 -18535.623,E2 -18535.623} C_VEL
LIN {X 0,Y 411.659,Z 807.759,A -85,B 0,C 180,E1 -18536.83,E2 -18536.83} C_VEL
LIN {X 0,Y 410.376,Z 814.585,A -85,B 0,C 180,E1 -18538.043,E2 -18538.043} C_VEL
LIN {X 0,Y 409.504,Z 819.283,A -85,B 0,C 180,E1 -18539.02,E2 -18539.02} C_VEL
LIN {X 0,Y 408.477,Z 825.019,A -85,B 0,C 180,E1 -18540.491,E2 -18540.491} C_VEL
LIN {X 0,Y 407.529,Z 829.573,A -85,B 0,C 180,E1 -18541.97,E2 -18541.97} C_VEL
LIN {X 0,Y 407.027,Z 833.097,A -85,B 0,C 180,E1 -18543.519,E2 -18543.519} C_VEL
LIN {X 0,Y 406.547,Z 835.385,A -85,B 0,C 180,E1 -18544.942,E2 -18544.942} C_VEL
LIN {X 0,Y 406.045,Z 836.961,A -85,B 0,C 180,E1 -18546.935,E2 -18546.935} C_VEL
LIN {X 0,Y 405.919,Z 837.228,A -85,B 0,C 180,E1 -18547.934,E2 -18547.934} C_VEL
LIN {X 0,Y 405.897,Z 836.203,A -85,B 0,C 180,E1 -18549.937,E2 -18549.937} C_VEL
LIN {X 0,Y 405.869,Z 835.125,A -85,B 0,C 180,E1 -18550.943,E2 -18550.943} C_VEL
LIN {X 0,Y 405.849,Z 832.545,A -85,B 0,C 180,E1 -18552.458,E2 -18552.458} C_VEL
LIN {X 0,Y 406.053,Z 828.859,A -85,B 0,C 180,E1 -18553.975,E2 -18553.975} C_VEL
LIN {X 0,Y 406.305,Z 822.908,A -85,B 0,C 180,E1 -18555.754,E2 -18555.754} C_VEL
LIN {X 0,Y 406.552,Z 817.525,A -85,B 0,C 180,E1 -18557.031,E2 -18557.031} C_VEL
LIN {X 0,Y 406.901,Z 811.234,A -85,B 0,C 180,E1 -18558.265,E2 -18558.265} C_VEL
LIN {X 0,Y 407.37,Z 803.004,A -85,B 0,C 180,E1 -18559.59,E2 -18559.59} C_VEL
LIN {X 0,Y 407.839,Z 794.328,A -85,B 0,C 180,E1 -18560.745,E2 -18560.745} C_VEL
LIN {X 0,Y 408.252,Z 786.328,A -85,B 0,C 180,E1 -18561.646,E2 -18561.646} C_VEL
LIN {X 0,Y 408.811,Z 776.819,A -85,B 0,C 180,E1 -18562.541,E2 -18562.541} C_VEL
LIN {X 0,Y 409.341,Z 766.933,A -85,B 0,C 180,E1 -18563.309,E2 -18563.309} C_VEL
LIN {X 0,Y 409.808,Z 756.788,A -85,B 0,C 180,E1 -18563.949,E2 -18563.949} C_VEL
LIN {X 0,Y 410.118,Z 745.608,A -85,B 0,C 180,E1 -18564.5,E2 -18564.5} C_VEL
LIN {X 0,Y 410.483,Z 735.231,A -85,B 0,C 180,E1 -18564.88,E2 -18564.88} C_VEL
LIN {X 0,Y 411.084,Z 714.261,A -85,B 0,C 180,E1 -18565.392,E2 -18565.392} C_VEL
LIN {X 0,Y 412.332,Z 653.679,A -85,B 0,C 180,E1 -18566.797,E2 -18566.797} C_VEL
LIN {X 0,Y 409.185,Z 627.749,A -85,B 0,C 180,E1 -18567.486,E2 -18567.486} C_VEL
LIN {X 0,Y 409.067,Z 626.356,A -85,B 0,C 180,E1 -18567.536,E2 -18567.536} C_VEL
LIN {X 0,Y 409.828,Z 615.215,A -85,B 0,C 180,E1 -18570.277,E2 -18570.277} C_VEL
LIN {X 0,Y 408.401,Z 606.543,A -85,B 0,C 180,E1 -18572.537,E2 -18572.537} C_VEL
LIN {X 0,Y 408.277,Z 606.561,A -85,B 0,C 180,E1 -18576.26,E2 -18576.26} C_VEL
LIN {X 0,Y 408.283,Z 606.557,A -85,B 0,C 180,E1 -18579.465,E2 -18579.465} C_VEL
LIN {X 0,Y 408.274,Z 606.559,A -85,B 0,C 180,E1 -18582.462,E2 -18582.462} C_VEL
LIN {X 0,Y 408.308,Z 606.553,A -85,B 0,C 180,E1 -18585.303,E2 -18585.303} C_VEL
LIN {X 0,Y 408.271,Z 606.565,A -85,B 0,C 180,E1 -18588.002,E2 -18588.002} C_VEL
LIN {X 0,Y 408.298,Z 606.555,A -85,B 0,C 180,E1 -18590.599,E2 -18590.599} C_VEL
LIN {X 0,Y 408.306,Z 606.557,A -85,B 0,C 180,E1 -18594.319,E2 -18594.319} C_VEL
LIN {X 0,Y 408.253,Z 606.565,A -85,B 0,C 180,E1 -18597.868,E2 -18597.868} C_VEL
LIN {X 0,Y 408.317,Z 606.552,A -85,B 0,C 180,E1 -18601.293,E2 -18601.293} C_VEL
LIN {X 0,Y 408.304,Z 606.554,A -85,B 0,C 180,E1 -18604.604,E2 -18604.604} C_VEL
LIN {X 0,Y 408.314,Z 606.558,A -85,B 0,C 180,E1 -18607.87,E2 -18607.87} C_VEL
LIN {X 0,Y 408.379,Z 606.544,A -85,B 0,C 180,E1 -18610.981,E2 -18610.981} C_VEL
LIN {X 0,Y 408.4,Z 606.548,A -85,B 0,C 180,E1 -18614.073,E2 -18614.073} C_VEL
LIN {X 0,Y 408.483,Z 606.536,A -85,B 0,C 180,E1 -18617.794,E2 -18617.794} C_VEL
LIN {X 0,Y 408.478,Z 606.532,A -85,B 0,C 180,E1 -18621.122,E2 -18621.122} C_VEL
LIN {X 0,Y 408.577,Z 606.526,A -85,B 0,C 180,E1 -18624.096,E2 -18624.096} C_VEL
LIN {X 0,Y 408.603,Z 606.516,A -85,B 0,C 180,E1 -18627.052,E2 -18627.052} C_VEL
LIN {X 0,Y 408.622,Z 606.521,A -85,B 0,C 180,E1 -18630,E2 -18630} C_VEL
LIN {X 0,Y 408.611,Z 606.522,A -85,B 0,C 180,E1 -18633.932,E2 -18633.932} C_VEL
LIN {X 0,Y 408.548,Z 606.523,A -85,B 0,C 180,E1 -18636.893,E2 -18636.893} C_VEL
LIN {X 0,Y 408.424,Z 606.544,A -85,B 0,C 180,E1 -18639.875,E2 -18639.875} C_VEL
LIN {X 0,Y 408.427,Z 606.538,A -85,B 0,C 180,E1 -18642.882,E2 -18642.882} C_VEL
LIN {X 0,Y 408.406,Z 606.546,A -85,B 0,C 180,E1 -18646.172,E2 -18646.172} C_VEL
LIN {X 0,Y 408.375,Z 606.545,A -85,B 0,C 180,E1 -18649.379,E2 -18649.379} C_VEL
LIN {X 0,Y 408.298,Z 606.554,A -85,B 0,C 180,E1 -18653.239,E2 -18653.239} C_VEL
LIN {X 0,Y 408.336,Z 606.551,A -85,B 0,C 180,E1 -18656.487,E2 -18656.487} C_VEL
LIN {X 0,Y 408.293,Z 606.56,A -85,B 0,C 180,E1 -18659.835,E2 -18659.835} C_VEL
LIN {X 0,Y 408.304,Z 606.554,A -85,B 0,C 180,E1 -18663.295,E2 -18663.295} C_VEL
LIN {X 0,Y 408.346,Z 606.552,A -85,B 0,C 180,E1 -18666.275,E2 -18666.275} C_VEL
LIN {X 0,Y 408.337,Z 606.551,A -85,B 0,C 180,E1 -18669.475,E2 -18669.475} C_VEL
LIN {X 0,Y 408.293,Z 606.555,A -85,B 0,C 180,E1 -18673.331,E2 -18673.331} C_VEL
LIN {X 0,Y 408.293,Z 606.555,A -85,B 0,C 180,E1 -18676.669,E2 -18676.669} C_VEL
LIN {X 0,Y 408.328,Z 606.551,A -85,B 0,C 180,E1 -18680.603,E2 -18680.603} C_VEL
LIN {X 0,Y 408.318,Z 606.555,A -85,B 0,C 180,E1 -18684.321,E2 -18684.321} C_VEL
LIN {X 0,Y 408.254,Z 606.565,A -85,B 0,C 180,E1 -18687.869,E2 -18687.869} C_VEL
LIN {X 0,Y 408.298,Z 606.554,A -85,B 0,C 180,E1 -18690.786,E2 -18690.786} C_VEL
LIN {X 0,Y 407.66,Z 606.638,A -85,B 0,C 180,E1 -18691.609,E2 -18691.609} C_VEL
LIN {X 0,Y 404.793,Z 606.991,A -85,B 0,C 180,E1 -18692.946,E2 -18692.946} C_VEL
LIN {X 0,Y 402.358,Z 607.301,A -85,B 0,C 180,E1 -18694.026,E2 -18694.026} C_VEL
LIN {X 0,Y 401.33,Z 607.423,A -85,B 0,C 180,E1 -18694.861,E2 -18694.861} C_VEL
LIN {X 0,Y 401.257,Z 607.431,A -85,B 0,C 180,E1 -18695.144,E2 -18695.144} C_VEL
LIN {X 0,Y 401.251,Z 607.434,A -85,B 0,C 180,E1 -18698.495,E2 -18698.495} C_VEL
LIN {X 0,Y 401.287,Z 607.431,A -85,B 0,C 180,E1 -18701.689,E2 -18701.689} C_VEL
LIN {X 0,Y 401.298,Z 607.426,A -85,B 0,C 180,E1 -18704.823,E2 -18704.823} C_VEL
LIN {X 0,Y 401.43,Z 607.416,A -85,B 0,C 180,E1 -18707.914,E2 -18707.914} C_VEL
LIN {X 0,Y 401.491,Z 607.409,A -85,B 0,C 180,E1 -18711.977,E2 -18711.977} C_VEL
LIN {X 0,Y 401.586,Z 607.398,A -85,B 0,C 180,E1 -18713.993,E2 -18713.993} C_VEL
LIN {X 0,Y 401.568,Z 607.392,A -85,B 0,C 180,E1 -18717.001,E2 -18717.001} C_VEL
LIN {X 0,Y 401.577,Z 607.399,A -85,B 0,C 180,E1 -18720,E2 -18720} C_VEL
LIN {X 0,Y 401.575,Z 607.399,A -85,B 0,C 180,E1 -18724.001,E2 -18724.001} C_VEL
LIN {X 0,Y 401.504,Z 607.4,A -85,B 0,C 180,E1 -18727.015,E2 -18727.015} C_VEL
LIN {X 0,Y 401.377,Z 607.423,A -85,B 0,C 180,E1 -18730.05,E2 -18730.05} C_VEL
LIN {X 0,Y 401.365,Z 607.418,A -85,B 0,C 180,E1 -18733.113,E2 -18733.113} C_VEL
LIN {X 0,Y 401.269,Z 607.434,A -85,B 0,C 180,E1 -18736.247,E2 -18736.247} C_VEL
LIN {X 0,Y 401.259,Z 607.433,A -85,B 0,C 180,E1 -18739.502,E2 -18739.502} C_VEL
LIN {X 0,Y 401.258,Z 607.432,A -85,B 0,C 180,E1 -18742.584,E2 -18742.584} C_VEL
LIN {X 0,Y 401.282,Z 607.434,A -85,B 0,C 180,E1 -18745.873,E2 -18745.873} C_VEL
LIN {X 0,Y 401.265,Z 607.431,A -85,B 0,C 180,E1 -18749.26,E2 -18749.26} C_VEL
LIN {X 0,Y 401.212,Z 607.437,A -85,B 0,C 180,E1 -18752.766,E2 -18752.766} C_VEL
